LIN {X 0,Y 466.236,Z 937.259,A -85,B 0,C 180,E1 20114.358,E2 20114.358} C_VEL
LIN {X 0,Y 461.421,Z 960.105,A -85,B 0,C 180,E1 20112.986,E2 20112.986} C_VEL
LIN {X 0,Y 456.989,Z 979.325,A -85,B 0,C 180,E1 20111.61,E2 20111.61} C_VEL
LIN {X 0,Y 451.374,Z 1001.605,A -85,B 0,C 180,E1 20109.724,E2 20109.724} C_VEL
LIN {X 0,Y 446.55,Z 1019.671,A -85,B 0,C 180,E1 20107.926,E2 20107.926} C_VEL
LIN {X 0,Y 441.064,Z 1039.324,A -85,B 0,C 180,E1 20105.635,E2 20105.635} C_VEL
LIN {X 0,Y 436.572,Z 1055.083,A -85,B 0,C 180,E1 20103.502,E2 20103.502} C_VEL
LIN {X 0,Y 431.661,Z 1072.275,A -85,B 0,C 180,E1 20100.792,E2 20100.792} C_VEL
LIN {X 0,Y 427.908,Z 1085.783,A -85,B 0,C 180,E1 20098.317,E2 20098.317} C_VEL
LIN {X 0,Y 424.121,Z 1100.061,A -85,B 0,C 180,E1 20095.26,E2 20095.26} C_VEL
LIN {X 0,Y 421.416,Z 1111.21,A -85,B 0,C 180,E1 20092.458,E2 20092.458} C_VEL
LIN {X 0,Y 419.039,Z 1122.409,A -85,B 0,C 180,E1 20089.105,E2 20089.105} C_VEL
LIN {X 0,Y 417.651,Z 1130.324,A -85,B 0,C 180,E1 20086.254,E2 20086.254} C_VEL
LIN {X 0,Y 416.596,Z 1138.166,A -85,B 0,C 180,E1 20082.757,E2 20082.757} C_VEL
LIN {X 0,Y 416.157,Z 1143.104,A -85,B 0,C 180,E1 20079.902,E2 20079.902} C_VEL
LIN {X 0,Y 415.971,Z 1147.181,A -85,B 0,C 180,E1 20076.764,E2 20076.764} C_VEL
LIN {X 0,Y 415.942,Z 1149.613,A -85,B 0,C 180,E1 20073.583,E2 20073.583} C_VEL
LIN {X 0,Y 415.943,Z 1150.522,A -85,B 0,C 180,E1 20070.964,E2 20070.964} C_VEL
LIN {X 0,Y 415.947,Z 1150.354,A -85,B 0,C 180,E1 20068.071,E2 20068.071} C_VEL
LIN {X 0,Y 415.927,Z 1148.612,A -85,B 0,C 180,E1 20064.897,E2 20064.897} C_VEL
LIN {X 0,Y 415.991,Z 1145.845,A -85,B 0,C 180,E1 20062.125,E2 20062.125} C_VEL
LIN {X 0,Y 416.258,Z 1141.713,A -85,B 0,C 180,E1 20059.201,E2 20059.201} C_VEL
LIN {X 0,Y 416.938,Z 1135.233,A -85,B 0,C 180,E1 20055.841,E2 20055.841} C_VEL
LIN {X 0,Y 417.947,Z 1128.442,A -85,B 0,C 180,E1 20053.03,E2 20053.03} C_VEL
LIN {X 0,Y 419.816,Z 1118.491,A -85,B 0,C 180,E1 20049.651,E2 20049.651} C_VEL
LIN {X 0,Y 422.069,Z 1108.405,A -85,B 0,C 180,E1 20046.807,E2 20046.807} C_VEL
LIN {X 0,Y 425.401,Z 1095.098,A -85,B 0,C 180,E1 20043.625,E2 20043.625} C_VEL
LIN {X 0,Y 428.676,Z 1082.856,A -85,B 0,C 180,E1 20041.129,E2 20041.129} C_VEL
LIN {X 0,Y 433.056,Z 1067.359,A -85,B 0,C 180,E1 20038.39,E2 20038.39} C_VEL
LIN {X 0,Y 437.389,Z 1052.082,A -85,B 0,C 180,E1 20036.082,E2 20036.082} C_VEL
LIN {X 0,Y 442.334,Z 1034.815,A -85,B 0,C 180,E1 20033.804,E2 20033.804} C_VEL
LIN {X 0,Y 447.361,Z 1016.456,A -85,B 0,C 180,E1 20031.748,E2 20031.748} C_VEL
LIN {X 0,Y 452.648,Z 996.689,A -85,B 0,C 180,E1 20029.832,E2 20029.832} C_VEL
LIN {X 0,Y 457.714,Z 976.039,A -85,B 0,C 180,E1 20028.153,E2 20028.153} C_VEL
LIN {X 0,Y 462.616,Z 954.653,A -85,B 0,C 180,E1 20026.667,E2 20026.667} C_VEL
LIN {X 0,Y 466.859,Z 933.595,A -85,B 0,C 180,E1 20025.459,E2 20025.459} C_VEL
LIN {X 0,Y 470.626,Z 912.697,A -85,B 0,C 180,E1 20024.449,E2 20024.449} C_VEL
LIN {X 0,Y 474.229,Z 888.902,A -85,B 0,C 180,E1 20023.533,E2 20023.533} C_VEL
LIN {X 0,Y 476.825,Z 868.071,A -85,B 0,C 180,E1 20022.903,E2 20022.903} C_VEL
LIN {X 0,Y 479.197,Z 841.622,A -85,B 0,C 180,E1 20022.311,E2 20022.311} C_VEL
LIN {X 0,Y 490.289,Z 617.268,A -85,B 0,C 180,E1 20018.698,E2 20018.698} C_VEL
LIN {X 0,Y 493.313,Z 555.727,A -85,B 0,C 180,E1 20017.706,E2 20017.706} C_VEL
LIN {X 0,Y 483.018,Z 538.654,A -85,B 0,C 180,E1 20015.789,E2 20015.789} C_VEL
LIN {X 0,Y 473.224,Z 523.488,A -85,B 0,C 180,E1 20013.832,E2 20013.832} C_VEL
LIN {X 0,Y 462.632,Z 508.305,A -85,B 0,C 180,E1 20011.536,E2 20011.536} C_VEL
LIN {X 0,Y 453.738,Z 496.412,A -85,B 0,C 180,E1 20009.434,E2 20009.434} C_VEL
LIN {X 0,Y 446.328,Z 486.795,A -85,B 0,C 180,E1 20007.52,E2 20007.52} C_VEL
LIN {X 0,Y 441.143,Z 480.531,A -85,B 0,C 180,E1 20006.086,E2 20006.086} C_VEL
LIN {X 0,Y 436.301,Z 474.731,A -85,B 0,C 180,E1 20004.652,E2 20004.652} C_VEL
LIN {X 0,Y 431.339,Z 468.954,A -85,B 0,C 180,E1 20003.064,E2 20003.064} C_VEL
LIN {X 0,Y 429.525,Z 465.262,A -85,B 0,C 180,E1 20001.724,E2 20001.724} C_VEL
LIN {X 0,Y 427.505,Z 461.609,A -85,B 0,C 180,E1 20000.11,E2 20000.11} C_VEL
LIN {X 0,Y 426.506,Z 459.96,A -85,B 0,C 180,E1 19999.303,E2 19999.303} C_VEL
LIN {X 0,Y 424.096,Z 455.355,A -85,B 0,C 180,E1 19996.999,E2 19996.999} C_VEL
LIN {X 0,Y 421.764,Z 451.295,A -85,B 0,C 180,E1 19994.554,E2 19994.554} C_VEL
LIN {X 0,Y 421.091,Z 450.043,A -85,B 0,C 180,E1 19993.736,E2 19993.736} C_VEL
LIN {X 0,Y 418.609,Z 445.587,A -85,B 0,C 180,E1 19990.181,E2 19990.181} C_VEL
LIN {X 0,Y 418.499,Z 445.082,A -85,B 0,C 180,E1 19988.657,E2 19988.657} C_VEL
LIN {X 0,Y 418.484,Z 445.068,A -85,B 0,C 180,E1 19984.897,E2 19984.897} C_VEL
LIN {X 0,Y 418.484,Z 445.066,A -85,B 0,C 180,E1 19981.095,E2 19981.095} C_VEL
LIN {X 0,Y 418.501,Z 445.072,A -85,B 0,C 180,E1 19977.398,E2 19977.398} C_VEL
LIN {X 0,Y 418.519,Z 445.085,A -85,B 0,C 180,E1 19973.553,E2 19973.553} C_VEL
LIN {X 0,Y 418.524,Z 445.143,A -85,B 0,C 180,E1 19969.678,E2 19969.678} C_VEL
LIN {X 0,Y 418.601,Z 445.836,A -85,B 0,C 180,E1 19968.704,E2 19968.704} C_VEL
LIN {X 0,Y 421.63,Z 451.075,A -85,B 0,C 180,E1 19964.597,E2 19964.597} C_VEL
LIN {X 0,Y 423.884,Z 455.148,A -85,B 0,C 180,E1 19962.142,E2 19962.142} C_VEL
LIN {X 0,Y 424.578,Z 456.381,A -85,B 0,C 180,E1 19961.462,E2 19961.462} C_VEL
LIN {X 0,Y 426.442,Z 459.915,A -85,B 0,C 180,E1 19959.695,E2 19959.695} C_VEL
LIN {X 0,Y 427.478,Z 462.022,A -85,B 0,C 180,E1 19958.743,E2 19958.743} C_VEL
LIN {X 0,Y 429.853,Z 466.303,A -85,B 0,C 180,E1 19956.851,E2 19956.851} C_VEL
LIN {X 0,Y 432.472,Z 471.575,A -85,B 0,C 180,E1 19954.823,E2 19954.823} C_VEL
LIN {X 0,Y 434.744,Z 476.119,A -85,B 0,C 180,E1 19953.205,E2 19953.205} C_VEL
LIN {X 0,Y 437.115,Z 481.055,A -85,B 0,C 180,E1 19951.589,E2 19951.589} C_VEL
LIN {X 0,Y 439.13,Z 484.762,A -85,B 0,C 180,E1 19950.502,E2 19950.502} C_VEL
LIN {X 0,Y 446.478,Z 494.703,A -85,B 0,C 180,E1 19948.434,E2 19948.434} C_VEL
LIN {X 0,Y 452.479,Z 502.886,A -85,B 0,C 180,E1 19946.885,E2 19946.885} C_VEL
LIN {X 0,Y 461.013,Z 515.147,A -85,B 0,C 180,E1 19944.841,E2 19944.841} C_VEL
LIN {X 0,Y 469.958,Z 528.922,A -85,B 0,C 180,E1 19942.864,E2 19942.864} C_VEL
LIN {X 0,Y 479.843,Z 544.931,A -85,B 0,C 180,E1 19940.847,E2 19940.847} C_VEL
LIN {X 0,Y 489.836,Z 562.594,A -85,B 0,C 180,E1 19938.945,E2 19938.945} C_VEL
LIN {X 0,Y 490.651,Z 564.525,A -85,B 0,C 180,E1 19938.786,E2 19938.786} C_VEL
LIN {X 0,Y 491.161,Z 569.373,A -85,B 0,C 180,E1 19938.607,E2 19938.607} C_VEL
LIN {X 0,Y 479.889,Z 824.745,A -85,B 0,C 180,E1 19934.734,E2 19934.734} C_VEL
LIN {X 0,Y 478.092,Z 855.335,A -85,B 0,C 180,E1 19934.21,E2 19934.21} C_VEL
LIN {X 0,Y 475.844,Z 877.482,A -85,B 0,C 180,E1 19933.668,E2 19933.668} C_VEL
LIN {X 0,Y 472.694,Z 900.618,A -85,B 0,C 180,E1 19932.891,E2 19932.891} C_VEL
LIN {X 0,Y 469.116,Z 922.276,A -85,B 0,C 180,E1 19931.966,E2 19931.966} C_VEL
LIN {X 0,Y 464.908,Z 943.457,A -85,B 0,C 180,E1 19930.831,E2 19930.831} C_VEL
LIN {X 0,Y 460.365,Z 963.847,A -85,B 0,C 180,E1 19929.523,E2 19929.523} C_VEL
LIN {X 0,Y 455.443,Z 983.36,A -85,B 0,C 180,E1 19928.003,E2 19928.003} C_VEL
LIN {X 0,Y 450.456,Z 1001.908,A -85,B 0,C 180,E1 19926.316,E2 19926.316} C_VEL
LIN {X 0,Y 445.221,Z 1019.736,A -85,B 0,C 180,E1 19924.38,E2 19924.38} C_VEL
LIN {X 0,Y 440.166,Z 1036.473,A -85,B 0,C 180,E1 19922.265,E2 19922.265} C_VEL
LIN {X 0,Y 435.489,Z 1051.384,A -85,B 0,C 180,E1 19920.035,E2 19920.035} C_VEL
LIN {X 0,Y 430.926,Z 1065.976,A -85,B 0,C 180,E1 19917.5,E2 19917.5} C_VEL
LIN {X 0,Y 427.066,Z 1078.461,A -85,B 0,C 180,E1 19914.925,E2 19914.925} C_VEL
LIN {X 0,Y 423.388,Z 1091.027,A -85,B 0,C 180,E1 19911.855,E2 19911.855} C_VEL
LIN {X 0,Y 420.871,Z 1100.299,A -85,B 0,C 180,E1 19909.139,E2 19909.139} C_VEL
LIN {X 0,Y 418.723,Z 1109.293,A -85,B 0,C 180,E1 19905.939,E2 19905.939} C_VEL
LIN {X 0,Y 417.417,Z 1115.919,A -85,B 0,C 180,E1 19903.013,E2 19903.013} C_VEL
LIN {X 0,Y 416.528,Z 1121.699,A -85,B 0,C 180,E1 19899.674,E2 19899.674} C_VEL
LIN {X 0,Y 416.151,Z 1125.344,A -85,B 0,C 180,E1 19896.761,E2 19896.761} C_VEL
LIN {X 0,Y 415.984,Z 1127.881,A -85,B 0,C 180,E1 19893.445,E2 19893.445} C_VEL
LIN {X 0,Y 415.96,Z 1128.751,A -85,B 0,C 180,E1 19890.689,E2 19890.689} C_VEL
LIN {X 0,Y 415.97,Z 1128.859,A -85,B 0,C 180,E1 19889.97,E2 19889.97} C_VEL
LIN {X 0,Y 414.938,Z 1128.793,A -85,B 0,C 180,E1 19888.908,E2 19888.908} C_VEL
LIN {X 0,Y 408.532,Z 1127.889,A -85,B 0,C 180,E1 19885.92,E2 19885.92} C_VEL
LIN {X 0,Y 408.028,Z 1127.363,A -85,B 0,C 180,E1 19885.143,E2 19885.143} C_VEL
LIN {X 0,Y 408.249,Z 1124.747,A -85,B 0,C 180,E1 19882.258,E2 19882.258} C_VEL
LIN {X 0,Y 408.8,Z 1120.397,A -85,B 0,C 180,E1 19879.002,E2 19879.002} C_VEL
LIN {X 0,Y 409.823,Z 1114.59,A -85,B 0,C 180,E1 19875.878,E2 19875.878} C_VEL
LIN {X 0,Y 411.56,Z 1106.902,A -85,B 0,C 180,E1 19872.613,E2 19872.613} C_VEL
LIN {X 0,Y 413.856,Z 1098.115,A -85,B 0,C 180,E1 19869.624,E2 19869.624} C_VEL
LIN {X 0,Y 417.224,Z 1086.65,A -85,B 0,C 180,E1 19866.408,E2 19866.408} C_VEL
LIN {X 0,Y 420.762,Z 1075.415,A -85,B 0,C 180,E1 19863.768,E2 19863.768} C_VEL
LIN {X 0,Y 425.294,Z 1061.422,A -85,B 0,C 180,E1 19860.997,E2 19860.997} C_VEL
LIN {X 0,Y 430.002,Z 1047.109,A -85,B 0,C 180,E1 19858.583,E2 19858.583} C_VEL
LIN {X 0,Y 435.22,Z 1030.861,A -85,B 0,C 180,E1 19856.271,E2 19856.271} C_VEL
LIN {X 0,Y 440.64,Z 1013.592,A -85,B 0,C 180,E1 19854.165,E2 19854.165} C_VEL
LIN {X 0,Y 446.057,Z 994.989,A -85,B 0,C 180,E1 19852.268,E2 19852.268} C_VEL
LIN {X 0,Y 451.521,Z 974.977,A -85,B 0,C 180,E1 19850.538,E2 19850.538} C_VEL
LIN {X 0,Y 456.076,Z 956.544,A -85,B 0,C 180,E1 19849.207,E2 19849.207} C_VEL
LIN {X 0,Y 460.892,Z 934.937,A -85,B 0,C 180,E1 19847.899,E2 19847.899} C_VEL
LIN {X 0,Y 464.708,Z 914.889,A -85,B 0,C 180,E1 19846.909,E2 19846.909} C_VEL
LIN {X 0,Y 468.44,Z 891.824,A -85,B 0,C 180,E1 19845.995,E2 19845.995} C_VEL
LIN {X 0,Y 471.082,Z 870.943,A -85,B 0,C 180,E1 19845.361,E2 19845.361} C_VEL
LIN {X 0,Y 473.346,Z 846.549,A -85,B 0,C 180,E1 19844.819,E2 19844.819} C_VEL
LIN {X 0,Y 481.939,Z 658.642,A -85,B 0,C 180,E1 19841.926,E2 19841.926} C_VEL
LIN {X 0,Y 486.071,Z 569.379,A -85,B 0,C 180,E1 19840.545,E2 19840.545} C_VEL
LIN {X 0,Y 485.457,Z 567.538,A -85,B 0,C 180,E1 19840.413,E2 19840.413} C_VEL
LIN {X 0,Y 475.186,Z 549.156,A -85,B 0,C 180,E1 19838.39,E2 19838.39} C_VEL
LIN {X 0,Y 463.604,Z 530.342,A -85,B 0,C 180,E1 19835.919,E2 19835.919} C_VEL
LIN {X 0,Y 451.846,Z 512.633,A -85,B 0,C 180,E1 19833.133,E2 19833.133} C_VEL
LIN {X 0,Y 445.276,Z 503.579,A -85,B 0,C 180,E1 19831.431,E2 19831.431} C_VEL
LIN {X 0,Y 438.875,Z 494.83,A -85,B 0,C 180,E1 19829.63,E2 19829.63} C_VEL
LIN {X 0,Y 434.964,Z 489.644,A -85,B 0,C 180,E1 19828.452,E2 19828.452} C_VEL
LIN {X 0,Y 429.781,Z 482.666,A -85,B 0,C 180,E1 19826.681,E2 19826.681} C_VEL
LIN {X 0,Y 428.07,Z 479.202,A -85,B 0,C 180,E1 19825.454,E2 19825.454} C_VEL
LIN {X 0,Y 426.124,Z 475.201,A -85,B 0,C 180,E1 19823.95,E2 19823.95} C_VEL
LIN {X 0,Y 423.943,Z 470.874,A -85,B 0,C 180,E1 19822.171,E2 19822.171} C_VEL
LIN {X 0,Y 421.585,Z 466.288,A -85,B 0,C 180,E1 19820.08,E2 19820.08} C_VEL
LIN {X 0,Y 419.645,Z 462.586,A -85,B 0,C 180,E1 19818.188,E2 19818.188} C_VEL
LIN {X 0,Y 416.217,Z 456.382,A -85,B 0,C 180,E1 19814.326,E2 19814.326} C_VEL
LIN {X 0,Y 413.397,Z 451.317,A -85,B 0,C 180,E1 19810.029,E2 19810.029} C_VEL
LIN {X 0,Y 410.952,Z 447.698,A -85,B 0,C 180,E1 19803.987,E2 19803.987} C_VEL
LIN {X 0,Y 410.734,Z 446.955,A -85,B 0,C 180,E1 19800.418,E2 19800.418} C_VEL
LIN {X 0,Y 410.903,Z 447.66,A -85,B 0,C 180,E1 19797.071,E2 19797.071} C_VEL
LIN {X 0,Y 412.969,Z 450.874,A -85,B 0,C 180,E1 19791.507,E2 19791.507} C_VEL
LIN {X 0,Y 413.909,Z 452.207,A -85,B 0,C 180,E1 19789.983,E2 19789.983} C_VEL
LIN {X 0,Y 416.606,Z 456.731,A -85,B 0,C 180,E1 19786.254,E2 19786.254} C_VEL
LIN {X 0,Y 419.083,Z 461.489,A -85,B 0,C 180,E1 19783.363,E2 19783.363} C_VEL
LIN {X 0,Y 420.011,Z 463.276,A -85,B 0,C 180,E1 19782.402,E2 19782.402} C_VEL
LIN {X 0,Y 422.459,Z 467.556,A -85,B 0,C 180,E1 19780.217,E2 19780.217} C_VEL
LIN {X 0,Y 423.625,Z 469.957,A -85,B 0,C 180,E1 19779.337,E2 19779.337} C_VEL
LIN {X 0,Y 427.225,Z 474.003,A -85,B 0,C 180,E1 19778.008,E2 19778.008} C_VEL
LIN {X 0,Y 432.384,Z 480.06,A -85,B 0,C 180,E1 19776.273,E2 19776.273} C_VEL
LIN {X 0,Y 436.767,Z 485.289,A -85,B 0,C 180,E1 19774.907,E2 19774.907} C_VEL
LIN {X 0,Y 441.245,Z 490.776,A -85,B 0,C 180,E1 19773.595,E2 19773.595} C_VEL
LIN {X 0,Y 446.228,Z 497.114,A -85,B 0,C 180,E1 19772.22,E2 19772.22} C_VEL
LIN {X 0,Y 454.022,Z 507.317,A -85,B 0,C 180,E1 19770.223,E2 19770.223} C_VEL
LIN {X 0,Y 463.425,Z 520.432,A -85,B 0,C 180,E1 19768.015,E2 19768.015} C_VEL
LIN {X 0,Y 474.721,Z 537.249,A -85,B 0,C 180,E1 19765.597,E2 19765.597} C_VEL
LIN {X 0,Y 487.154,Z 557.652,A -85,B 0,C 180,E1 19763.159,E2 19763.159} C_VEL
LIN {X 0,Y 488.226,Z 559.815,A -85,B 0,C 180,E1 19762.951,E2 19762.951} C_VEL
LIN {X 0,Y 476.442,Z 790.275,A -85,B 0,C 180,E1 19759.246,E2 19759.246} C_VEL
LIN {X 0,Y 473.431,Z 846.64,A -85,B 0,C 180,E1 19758.306,E2 19758.306} C_VEL
LIN {X 0,Y 470.957,Z 870.988,A -85,B 0,C 180,E1 19757.723,E2 19757.723} C_VEL
LIN {X 0,Y 467.992,Z 893.628,A -85,B 0,C 180,E1 19757.011,E2 19757.011} C_VEL
LIN {X 0,Y 464.181,Z 916.79,A -85,B 0,C 180,E1 19756.064,E2 19756.064} C_VEL
LIN {X 0,Y 460.216,Z 937.876,A -85,B 0,C 180,E1 19755.008,E2 19755.008} C_VEL
LIN {X 0,Y 455.197,Z 960.834,A -85,B 0,C 180,E1 19753.61,E2 19753.61} C_VEL
LIN {X 0,Y 450.466,Z 980.654,A -85,B 0,C 180,E1 19752.171,E2 19752.171} C_VEL
LIN {X 0,Y 444.882,Z 1001.936,A -85,B 0,C 180,E1 19750.338,E2 19750.338} C_VEL
LIN {X 0,Y 439.892,Z 1019.961,A -85,B 0,C 180,E1 19748.522,E2 19748.522} C_VEL
LIN {X 0,Y 434.358,Z 1039.027,A -85,B 0,C 180,E1 19746.272,E2 19746.272} C_VEL
LIN {X 0,Y 429.514,Z 1055.379,A -85,B 0,C 180,E1 19744.029,E2 19744.029} C_VEL
LIN {X 0,Y 424.544,Z 1072.008,A -85,B 0,C 180,E1 19741.366,E2 19741.366} C_VEL
LIN {X 0,Y 420.613,Z 1085.524,A -85,B 0,C 180,E1 19738.854,E2 19738.854} C_VEL
LIN {X 0,Y 416.631,Z 1099.816,A -85,B 0,C 180,E1 19735.747,E2 19735.747} C_VEL
LIN {X 0,Y 413.783,Z 1110.97,A -85,B 0,C 180,E1 19732.896,E2 19732.896} C_VEL
LIN {X 0,Y 411.246,Z 1122.249,A -85,B 0,C 180,E1 19729.457,E2 19729.457} C_VEL
LIN {X 0,Y 409.785,Z 1130.065,A -85,B 0,C 180,E1 19726.588,E2 19726.588} C_VEL
LIN {X 0,Y 408.651,Z 1137.946,A -85,B 0,C 180,E1 19723.009,E2 19723.009} C_VEL
LIN {X 0,Y 408.18,Z 1142.796,A -85,B 0,C 180,E1 19720.159,E2 19720.159} C_VEL
LIN {X 0,Y 407.982,Z 1146.872,A -85,B 0,C 180,E1 19716.98,E2 19716.98} C_VEL
LIN {X 0,Y 407.946,Z 1149.331,A -85,B 0,C 180,E1 19713.795,E2 19713.795} C_VEL
LIN {X 0,Y 407.95,Z 1150.289,A -85,B 0,C 180,E1 19711.124,E2 19711.124} C_VEL
LIN {X 0,Y 407.95,Z 1150.216,A -85,B 0,C 180,E1 19708.455,E2 19708.455} C_VEL
LIN {X 0,Y 407.934,Z 1148.754,A -85,B 0,C 180,E1 19705.22,E2 19705.22} C_VEL
LIN {X 0,Y 407.982,Z 1145.962,A -85,B 0,C 180,E1 19702.253,E2 19702.253} C_VEL
LIN {X 0,Y 408.228,Z 1142.139,A -85,B 0,C 180,E1 19699.415,E2 19699.415} C_VEL
LIN {X 0,Y 408.9,Z 1135.95,A -85,B 0,C 180,E1 19695.99,E2 19695.99} C_VEL
LIN {X 0,Y 409.979,Z 1128.861,A -85,B 0,C 180,E1 19692.949,E2 19692.949} C_VEL
LIN {X 0,Y 411.794,Z 1119.671,A -85,B 0,C 180,E1 19689.682,E2 19689.682} C_VEL
LIN {X 0,Y 414.17,Z 1109.348,A -85,B 0,C 180,E1 19686.676,E2 19686.676} C_VEL
LIN {X 0,Y 417.349,Z 1097.231,A -85,B 0,C 180,E1 19683.642,E2 19683.642} C_VEL
LIN {X 0,Y 421.006,Z 1084.029,A -85,B 0,C 180,E1 19680.864,E2 19680.864} C_VEL
LIN {X 0,Y 425.266,Z 1069.575,A -85,B 0,C 180,E1 19678.219,E2 19678.219} C_VEL
LIN {X 0,Y 430.084,Z 1053.293,A -85,B 0,C 180,E1 19675.682,E2 19675.682} C_VEL
LIN {X 0,Y 434.968,Z 1036.862,A -85,B 0,C 180,E1 19673.46,E2 19673.46} C_VEL
LIN {X 0,Y 440.387,Z 1017.978,A -85,B 0,C 180,E1 19671.28,E2 19671.28} C_VEL
LIN {X 0,Y 445.24,Z 1000.431,A -85,B 0,C 180,E1 19669.532,E2 19669.532} C_VEL
LIN {X 0,Y 450.867,Z 978.743,A -85,B 0,C 180,E1 19667.695,E2 19667.695} C_VEL
LIN {X 0,Y 455.394,Z 959.724,A -85,B 0,C 180,E1 19666.327,E2 19666.327} C_VEL
LIN {X 0,Y 460.414,Z 936.48,A -85,B 0,C 180,E1 19664.929,E2 19664.929} C_VEL
LIN {X 0,Y 464.258,Z 915.95,A -85,B 0,C 180,E1 19663.908,E2 19663.908} C_VEL
LIN {X 0,Y 468.237,Z 891.258,A -85,B 0,C 180,E1 19662.919,E2 19662.919} C_VEL
LIN {X 0,Y 470.981,Z 870.101,A -85,B 0,C 180,E1 19662.263,E2 19662.263} C_VEL
LIN {X 0,Y 473.431,Z 845.26,A -85,B 0,C 180,E1 19661.679,E2 19661.679} C_VEL
LIN {X 0,Y 477.17,Z 773.846,A -85,B 0,C 180,E1 19660.498,E2 19660.498} C_VEL
LIN {X 0,Y 488.114,Z 559.467,A -85,B 0,C 180,E1 19657.05,E2 19657.05} C_VEL
LIN {X 0,Y 476.77,Z 540.614,A -85,B 0,C 180,E1 19654.855,E2 19654.855} C_VEL
LIN {X 0,Y 466.825,Z 525.484,A -85,B 0,C 180,E1 19652.777,E2 19652.777} C_VEL
LIN {X 0,Y 456.774,Z 511.022,A -85,B 0,C 180,E1 19650.485,E2 19650.485} C_VEL
LIN {X 0,Y 447.495,Z 498.7,A -85,B 0,C 180,E1 19648.166,E2 19648.166} C_VEL
LIN {X 0,Y 439.334,Z 488.324,A -85,B 0,C 180,E1 19645.911,E2 19645.911} C_VEL
LIN {X 0,Y 433.643,Z 481.552,A -85,B 0,C 180,E1 19644.196,E2 19644.196} C_VEL
LIN {X 0,Y 428.84,Z 475.886,A -85,B 0,C 180,E1 19642.626,E2 19642.626} C_VEL
LIN {X 0,Y 425.089,Z 471.586,A -85,B 0,C 180,E1 19641.31,E2 19641.31} C_VEL
LIN {X 0,Y 422.894,Z 468.789,A -85,B 0,C 180,E1 19640.339,E2 19640.339} C_VEL
LIN {X 0,Y 421.848,Z 466.525,A -85,B 0,C 180,E1 19639.375,E2 19639.375} C_VEL
LIN {X 0,Y 419.726,Z 462.397,A -85,B 0,C 180,E1 19637.324,E2 19637.324} C_VEL
LIN {X 0,Y 416.96,Z 457.656,A -85,B 0,C 180,E1 19634.442,E2 19634.442} C_VEL
LIN {X 0,Y 416.288,Z 456.416,A -85,B 0,C 180,E1 19633.615,E2 19633.615} C_VEL
LIN {X 0,Y 413.474,Z 451.36,A -85,B 0,C 180,E1 19629.465,E2 19629.465} C_VEL
LIN {X 0,Y 410.866,Z 447.487,A -85,B 0,C 180,E1 19623.348,E2 19623.348} C_VEL
LIN {X 0,Y 410.683,Z 446.579,A -85,B 0,C 180,E1 19619.86,E2 19619.86} C_VEL
LIN {X 0,Y 410.796,Z 447.248,A -85,B 0,C 180,E1 19616.232,E2 19616.232} C_VEL
LIN {X 0,Y 412.43,Z 450.304,A -85,B 0,C 180,E1 19611.074,E2 19611.074} C_VEL
LIN {X 0,Y 413.759,Z 451.952,A -85,B 0,C 180,E1 19608.994,E2 19608.994} C_VEL
LIN {X 0,Y 416.829,Z 457.521,A -85,B 0,C 180,E1 19604.649,E2 19604.649} C_VEL
LIN {X 0,Y 419.209,Z 461.669,A -85,B 0,C 180,E1 19602.08,E2 19602.08} C_VEL
LIN {X 0,Y 421.569,Z 466.252,A -85,B 0,C 180,E1 19599.739,E2 19599.739} C_VEL
LIN {X 0,Y 424.757,Z 472.41,A -85,B 0,C 180,E1 19596.989,E2 19596.989} C_VEL
LIN {X 0,Y 427.331,Z 477.665,A -85,B 0,C 180,E1 19594.943,E2 19594.943} C_VEL
LIN {X 0,Y 429.595,Z 482.246,A -85,B 0,C 180,E1 19593.307,E2 19593.307} C_VEL
LIN {X 0,Y 431.567,Z 485.164,A -85,B 0,C 180,E1 19592.469,E2 19592.469} C_VEL
LIN {X 0,Y 437.443,Z 493.007,A -85,B 0,C 180,E1 19590.64,E2 19590.64} C_VEL
LIN {X 0,Y 443.691,Z 501.448,A -85,B 0,C 180,E1 19588.856,E2 19588.856} C_VEL
LIN {X 0,Y 449.505,Z 509.486,A -85,B 0,C 180,E1 19587.318,E2 19587.318} C_VEL
LIN {X 0,Y 458.139,Z 522.121,A -85,B 0,C 180,E1 19585.199,E2 19585.199} C_VEL
LIN {X 0,Y 466.687,Z 535.452,A -85,B 0,C 180,E1 19583.267,E2 19583.267} C_VEL
LIN {X 0,Y 476.309,Z 551.29,A -85,B 0,C 180,E1 19581.256,E2 19581.256} C_VEL
LIN {X 0,Y 485.816,Z 568.322,A -85,B 0,C 180,E1 19579.4,E2 19579.4} C_VEL
LIN {X 0,Y 485.988,Z 571.508,A -85,B 0,C 180,E1 19579.303,E2 19579.303} C_VEL
LIN {X 0,Y 474.351,Z 825.865,A -85,B 0,C 180,E1 19575.418,E2 19575.418} C_VEL
LIN {X 0,Y 472.525,Z 855.575,A -85,B 0,C 180,E1 19574.903,E2 19574.903} C_VEL
LIN {X 0,Y 470.2,Z 877.799,A -85,B 0,C 180,E1 19574.355,E2 19574.355} C_VEL
LIN {X 0,Y 467.002,Z 900.564,A -85,B 0,C 180,E1 19573.585,E2 19573.585} C_VEL
LIN {X 0,Y 463.329,Z 922.167,A -85,B 0,C 180,E1 19572.659,E2 19572.659} C_VEL
LIN {X 0,Y 459.017,Z 943.271,A -85,B 0,C 180,E1 19571.524,E2 19571.524} C_VEL
LIN {X 0,Y 454.345,Z 963.629,A -85,B 0,C 180,E1 19570.212,E2 19570.212} C_VEL
LIN {X 0,Y 449.331,Z 982.931,A -85,B 0,C 180,E1 19568.705,E2 19568.705} C_VEL
LIN {X 0,Y 444.041,Z 1001.994,A -85,B 0,C 180,E1 19566.958,E2 19566.958} C_VEL
LIN {X 0,Y 438.58,Z 1019.974,A -85,B 0,C 180,E1 19564.986,E2 19564.986} C_VEL
LIN {X 0,Y 433.312,Z 1036.753,A -85,B 0,C 180,E1 19562.839,E2 19562.839} C_VEL
LIN {X 0,Y 428.366,Z 1051.938,A -85,B 0,C 180,E1 19560.535,E2 19560.535} C_VEL
LIN {X 0,Y 423.475,Z 1066.914,A -85,B 0,C 180,E1 19557.873,E2 19557.873} C_VEL
LIN {X 0,Y 419.677,Z 1078.709,A -85,B 0,C 180,E1 19555.395,E2 19555.395} C_VEL
LIN {X 0,Y 415.878,Z 1091.075,A -85,B 0,C 180,E1 19552.326,E2 19552.326} C_VEL
LIN {X 0,Y 413.18,Z 1100.531,A -85,B 0,C 180,E1 19549.509,E2 19549.509} C_VEL
LIN {X 0,Y 410.909,Z 1109.518,A -85,B 0,C 180,E1 19546.251,E2 19546.251} C_VEL
LIN {X 0,Y 409.521,Z 1116.14,A -85,B 0,C 180,E1 19543.268,E2 19543.268} C_VEL
LIN {X 0,Y 408.575,Z 1121.915,A -85,B 0,C 180,E1 19539.864,E2 19539.864} C_VEL
LIN {X 0,Y 408.167,Z 1125.558,A -85,B 0,C 180,E1 19536.894,E2 19536.894} C_VEL
LIN {X 0,Y 407.988,Z 1128.092,A -85,B 0,C 180,E1 19533.513,E2 19533.513} C_VEL
LIN {X 0,Y 407.963,Z 1128.961,A -85,B 0,C 180,E1 19530.702,E2 19530.702} C_VEL
LIN {X 0,Y 407.972,Z 1128.596,A -85,B 0,C 180,E1 19527.472,E2 19527.472} C_VEL
LIN {X 0,Y 408.028,Z 1127.363,A -85,B 0,C 180,E1 19525.143,E2 19525.143} C_VEL
LIN {X 0,Y 407.087,Z 1126.577,A -85,B 0,C 180,E1 19524.066,E2 19524.066} C_VEL
LIN {X 0,Y 400.941,Z 1123.752,A -85,B 0,C 180,E1 19521.035,E2 19521.035} C_VEL
LIN {X 0,Y 400.541,Z 1122.704,A -85,B 0,C 180,E1 19520.252,E2 19520.252} C_VEL
LIN {X 0,Y 401.391,Z 1117.669,A -85,B 0,C 180,E1 19517.044,E2 19517.044} C_VEL
LIN {X 0,Y 402.89,Z 1110.666,A -85,B 0,C 180,E1 19513.713,E2 19513.713} C_VEL
LIN {X 0,Y 405.078,Z 1102.402,A -85,B 0,C 180,E1 19510.535,E2 19510.535} C_VEL
LIN {X 0,Y 407.934,Z 1092.652,A -85,B 0,C 180,E1 19507.519,E2 19507.519} C_VEL
LIN {X 0,Y 411.619,Z 1081.236,A -85,B 0,C 180,E1 19504.535,E2 19504.535} C_VEL
LIN {X 0,Y 415.681,Z 1069.001,A -85,B 0,C 180,E1 19501.87,E2 19501.87} C_VEL
LIN {X 0,Y 420.508,Z 1054.969,A -85,B 0,C 180,E1 19499.254,E2 19499.254} C_VEL
LIN {X 0,Y 425.415,Z 1040.367,A -85,B 0,C 180,E1 19496.955,E2 19496.955} C_VEL
LIN {X 0,Y 430.931,Z 1023.738,A -85,B 0,C 180,E1 19494.707,E2 19494.707} C_VEL
LIN {X 0,Y 436.28,Z 1006.72,A -85,B 0,C 180,E1 19492.767,E2 19492.767} C_VEL
LIN {X 0,Y 442.081,Z 987.161,A -85,B 0,C 180,E1 19490.873,E2 19490.873} C_VEL
LIN {X 0,Y 447.016,Z 968.938,A -85,B 0,C 180,E1 19489.389,E2 19489.389} C_VEL
LIN {X 0,Y 452.393,Z 947.06,A -85,B 0,C 180,E1 19487.902,E2 19487.902} C_VEL
LIN {X 0,Y 456.631,Z 927.356,A -85,B 0,C 180,E1 19486.797,E2 19486.797} C_VEL
LIN {X 0,Y 460.923,Z 903.891,A -85,B 0,C 180,E1 19485.735,E2 19485.735} C_VEL
LIN {X 0,Y 464.19,Z 882.173,A -85,B 0,C 180,E1 19484.965,E2 19484.965} C_VEL
LIN {X 0,Y 466.866,Z 858.532,A -85,B 0,C 180,E1 19484.346,E2 19484.346} C_VEL
LIN {X 0,Y 468.623,Z 834.837,A -85,B 0,C 180,E1 19483.901,E2 19483.901} C_VEL
LIN {X 0,Y 480.564,Z 582.416,A -85,B 0,C 180,E1 19480.02,E2 19480.02} C_VEL
LIN {X 0,Y 480.926,Z 572.23,A -85,B 0,C 180,E1 19479.841,E2 19479.841} C_VEL
LIN {X 0,Y 470.994,Z 554.364,A -85,B 0,C 180,E1 19477.826,E2 19477.826} C_VEL
LIN {X 0,Y 460.328,Z 536.752,A -85,B 0,C 180,E1 19475.486,E2 19475.486} C_VEL
LIN {X 0,Y 448.855,Z 519.233,A -85,B 0,C 180,E1 19472.698,E2 19472.698} C_VEL
LIN {X 0,Y 442.183,Z 509.916,A -85,B 0,C 180,E1 19470.922,E2 19470.922} C_VEL
LIN {X 0,Y 436.194,Z 501.605,A -85,B 0,C 180,E1 19469.189,E2 19469.189} C_VEL
LIN {X 0,Y 432.346,Z 496.463,A -85,B 0,C 180,E1 19468.001,E2 19468.001} C_VEL
LIN {X 0,Y 425.315,Z 487.258,A -85,B 0,C 180,E1 19465.631,E2 19465.631} C_VEL
LIN {X 0,Y 421.448,Z 481.892,A -85,B 0,C 180,E1 19464.084,E2 19464.084} C_VEL
LIN {X 0,Y 418.669,Z 476.691,A -85,B 0,C 180,E1 19461.874,E2 19461.874} C_VEL
LIN {X 0,Y 416.571,Z 472.463,A -85,B 0,C 180,E1 19459.928,E2 19459.928} C_VEL
LIN {X 0,Y 414.666,Z 468.658,A -85,B 0,C 180,E1 19457.978,E2 19457.978} C_VEL
LIN {X 0,Y 411.401,Z 462.741,A -85,B 0,C 180,E1 19454.21,E2 19454.21} C_VEL
LIN {X 0,Y 408.732,Z 457.814,A -85,B 0,C 180,E1 19450.002,E2 19450.002} C_VEL
LIN {X 0,Y 406.344,Z 454.233,A -85,B 0,C 180,E1 19443.951,E2 19443.951} C_VEL
LIN {X 0,Y 406.121,Z 453.472,A -85,B 0,C 180,E1 19440.282,E2 19440.282} C_VEL
LIN {X 0,Y 406.337,Z 454.287,A -85,B 0,C 180,E1 19436.897,E2 19436.897} C_VEL
LIN {X 0,Y 408.501,Z 457.578,A -85,B 0,C 180,E1 19431.271,E2 19431.271} C_VEL
LIN {X 0,Y 409.28,Z 458.943,A -85,B 0,C 180,E1 19429.869,E2 19429.869} C_VEL
LIN {X 0,Y 412.108,Z 463.755,A -85,B 0,C 180,E1 19425.958,E2 19425.958} C_VEL
LIN {X 0,Y 414.261,Z 467.843,A -85,B 0,C 180,E1 19423.452,E2 19423.452} C_VEL
LIN {X 0,Y 415.313,Z 470,A -85,B 0,C 180,E1 19422.341,E2 19422.341} C_VEL
LIN {X 0,Y 420.097,Z 475.511,A -85,B 0,C 180,E1 19420.246,E2 19420.246} C_VEL
LIN {X 0,Y 425.52,Z 481.795,A -85,B 0,C 180,E1 19418.206,E2 19418.206} C_VEL
LIN {X 0,Y 430.443,Z 487.655,A -85,B 0,C 180,E1 19416.523,E2 19416.523} C_VEL
LIN {X 0,Y 434.484,Z 492.553,A -85,B 0,C 180,E1 19415.238,E2 19415.238} C_VEL
LIN {X 0,Y 438.9,Z 498.053,A -85,B 0,C 180,E1 19413.916,E2 19413.916} C_VEL
LIN {X 0,Y 445.993,Z 507.122,A -85,B 0,C 180,E1 19411.95,E2 19411.95} C_VEL
LIN {X 0,Y 455.777,Z 520.504,A -85,B 0,C 180,E1 19409.478,E2 19409.478} C_VEL
LIN {X 0,Y 467.282,Z 537.414,A -85,B 0,C 180,E1 19406.858,E2 19406.858} C_VEL
LIN {X 0,Y 478.916,Z 556.153,A -85,B 0,C 180,E1 19404.447,E2 19404.447} C_VEL
LIN {X 0,Y 483.029,Z 563.567,A -85,B 0,C 180,E1 19403.632,E2 19403.632} C_VEL
LIN {X 0,Y 470.93,Z 793.043,A -85,B 0,C 180,E1 19399.921,E2 19399.921} C_VEL
LIN {X 0,Y 467.945,Z 846.962,A -85,B 0,C 180,E1 19399.014,E2 19399.014} C_VEL
LIN {X 0,Y 465.4,Z 871.25,A -85,B 0,C 180,E1 19398.428,E2 19398.428} C_VEL
LIN {X 0,Y 462.317,Z 894.124,A -85,B 0,C 180,E1 19397.704,E2 19397.704} C_VEL
LIN {X 0,Y 458.43,Z 916.982,A -85,B 0,C 180,E1 19396.761,E2 19396.761} C_VEL
LIN {X 0,Y 454.483,Z 937.356,A -85,B 0,C 180,E1 19395.735,E2 19395.735} C_VEL
LIN {X 0,Y 449.311,Z 960.408,A -85,B 0,C 180,E1 19394.329,E2 19394.329} C_VEL
LIN {X 0,Y 444.646,Z 979.355,A -85,B 0,C 180,E1 19392.951,E2 19392.951} C_VEL
LIN {X 0,Y 438.833,Z 1000.915,A -85,B 0,C 180,E1 19391.099,E2 19391.099} C_VEL
LIN {X 0,Y 433.636,Z 1019.017,A -85,B 0,C 180,E1 19389.268,E2 19389.268} C_VEL
LIN {X 0,Y 427.654,Z 1038.906,A -85,B 0,C 180,E1 19386.905,E2 19386.905} C_VEL
LIN {X 0,Y 422.838,Z 1054.513,A -85,B 0,C 180,E1 19384.743,E2 19384.743} C_VEL
LIN {X 0,Y 417.475,Z 1071.744,A -85,B 0,C 180,E1 19381.959,E2 19381.959} C_VEL
LIN {X 0,Y 413.354,Z 1085.266,A -85,B 0,C 180,E1 19379.41,E2 19379.41} C_VEL
LIN {X 0,Y 409.173,Z 1099.572,A -85,B 0,C 180,E1 19376.251,E2 19376.251} C_VEL
LIN {X 0,Y 406.307,Z 1110.202,A -85,B 0,C 180,E1 19373.495,E2 19373.495} C_VEL
LIN {X 0,Y 403.577,Z 1121.601,A -85,B 0,C 180,E1 19369.993,E2 19369.993} C_VEL
LIN {X 0,Y 401.984,Z 1129.474,A -85,B 0,C 180,E1 19367.068,E2 19367.068} C_VEL
LIN {X 0,Y 400.822,Z 1136.936,A -85,B 0,C 180,E1 19363.709,E2 19363.709} C_VEL
LIN {X 0,Y 400.216,Z 1142.365,A -85,B 0,C 180,E1 19360.509,E2 19360.509} C_VEL
LIN {X 0,Y 399.976,Z 1146.258,A -85,B 0,C 180,E1 19357.469,E2 19357.469} C_VEL
LIN {X 0,Y 399.949,Z 1149.05,A -85,B 0,C 180,E1 19354.014,E2 19354.014} C_VEL
LIN {X 0,Y 399.953,Z 1150.079,A -85,B 0,C 180,E1 19351.146,E2 19351.146} C_VEL
LIN {X 0,Y 399.952,Z 1150.006,A -85,B 0,C 180,E1 19348.424,E2 19348.424} C_VEL
LIN {X 0,Y 399.933,Z 1148.542,A -85,B 0,C 180,E1 19345.124,E2 19345.124} C_VEL
LIN {X 0,Y 399.992,Z 1145.748,A -85,B 0,C 180,E1 19342.097,E2 19342.097} C_VEL
LIN {X 0,Y 400.256,Z 1141.922,A -85,B 0,C 180,E1 19339.201,E2 19339.201} C_VEL
LIN {X 0,Y 400.973,Z 1135.726,A -85,B 0,C 180,E1 19335.707,E2 19335.707} C_VEL
LIN {X 0,Y 402.113,Z 1128.716,A -85,B 0,C 180,E1 19332.639,E2 19332.639} C_VEL
LIN {X 0,Y 404.039,Z 1119.519,A -85,B 0,C 180,E1 19329.302,E2 19329.302} C_VEL
LIN {X 0,Y 406.609,Z 1108.969,A -85,B 0,C 180,E1 19326.176,E2 19326.176} C_VEL
LIN {X 0,Y 410.053,Z 1096.542,A -85,B 0,C 180,E1 19323.028,E2 19323.028} C_VEL
LIN {X 0,Y 413.982,Z 1083.05,A -85,B 0,C 180,E1 19320.162,E2 19320.162} C_VEL
LIN {X 0,Y 418.496,Z 1068.513,A -85,B 0,C 180,E1 19317.481,E2 19317.481} C_VEL
LIN {X 0,Y 423.542,Z 1052.058,A -85,B 0,C 180,E1 19314.911,E2 19314.911} C_VEL
LIN {X 0,Y 428.996,Z 1034.461,A -85,B 0,C 180,E1 19312.531,E2 19312.531} C_VEL
LIN {X 0,Y 434.522,Z 1015.79,A -85,B 0,C 180,E1 19310.401,E2 19310.401} C_VEL
LIN {X 0,Y 440.203,Z 995.934,A -85,B 0,C 180,E1 19308.451,E2 19308.451} C_VEL
LIN {X 0,Y 445.454,Z 975.874,A -85,B 0,C 180,E1 19306.794,E2 19306.794} C_VEL
LIN {X 0,Y 450.636,Z 954.701,A -85,B 0,C 180,E1 19305.301,E2 19305.301} C_VEL
LIN {X 0,Y 455.367,Z 932.526,A -85,B 0,C 180,E1 19304.018,E2 19304.018} C_VEL
LIN {X 0,Y 459.649,Z 910.042,A -85,B 0,C 180,E1 19302.936,E2 19302.936} C_VEL
LIN {X 0,Y 463.244,Z 886.964,A -85,B 0,C 180,E1 19302.066,E2 19302.066} C_VEL
LIN {X 0,Y 466.142,Z 864.59,A -85,B 0,C 180,E1 19301.401,E2 19301.401} C_VEL
LIN {X 0,Y 468.317,Z 839.93,A -85,B 0,C 180,E1 19300.868,E2 19300.868} C_VEL
LIN {X 0,Y 480.437,Z 609.562,A -85,B 0,C 180,E1 19297.117,E2 19297.117} C_VEL
LIN {X 0,Y 482.849,Z 562.986,A -85,B 0,C 180,E1 19296.354,E2 19296.354} C_VEL
LIN {X 0,Y 470.765,Z 542.94,A -85,B 0,C 180,E1 19293.923,E2 19293.923} C_VEL
LIN {X 0,Y 459.996,Z 526.693,A -85,B 0,C 180,E1 19291.559,E2 19291.559} C_VEL
LIN {X 0,Y 450.519,Z 513.282,A -85,B 0,C 180,E1 19289.276,E2 19289.276} C_VEL
LIN {X 0,Y 441.131,Z 500.813,A -85,B 0,C 180,E1 19286.776,E2 19286.776} C_VEL
LIN {X 0,Y 435.69,Z 494.092,A -85,B 0,C 180,E1 19285.196,E2 19285.196} C_VEL
LIN {X 0,Y 431.496,Z 488.9,A -85,B 0,C 180,E1 19283.888,E2 19283.888} C_VEL
LIN {X 0,Y 426.575,Z 483.038,A -85,B 0,C 180,E1 19282.244,E2 19282.244} C_VEL
LIN {X 0,Y 422.889,Z 478.768,A -85,B 0,C 180,E1 19280.918,E2 19280.918} C_VEL
LIN {X 0,Y 418.279,Z 473.501,A -85,B 0,C 180,E1 19279.117,E2 19279.117} C_VEL
LIN {X 0,Y 415.226,Z 469.78,A -85,B 0,C 180,E1 19277.663,E2 19277.663} C_VEL
LIN {X 0,Y 414.275,Z 467.871,A -85,B 0,C 180,E1 19276.692,E2 19276.692} C_VEL
LIN {X 0,Y 412.086,Z 463.747,A -85,B 0,C 180,E1 19274.186,E2 19274.186} C_VEL
LIN {X 0,Y 408.822,Z 457.866,A -85,B 0,C 180,E1 19269.431,E2 19269.431} C_VEL
LIN {X 0,Y 406.255,Z 454,A -85,B 0,C 180,E1 19263.245,E2 19263.245} C_VEL
LIN {X 0,Y 406.02,Z 453.093,A -85,B 0,C 180,E1 19259.718,E2 19259.718} C_VEL
LIN {X 0,Y 406.222,Z 453.852,A -85,B 0,C 180,E1 19256.048,E2 19256.048} C_VEL
LIN {X 0,Y 408.694,Z 457.75,A -85,B 0,C 180,E1 19249.712,E2 19249.712} C_VEL
LIN {X 0,Y 411.974,Z 463.78,A -85,B 0,C 180,E1 19244.804,E2 19244.804} C_VEL
LIN {X 0,Y 414.355,Z 468.011,A -85,B 0,C 180,E1 19242.153,E2 19242.153} C_VEL
LIN {X 0,Y 416.7,Z 472.593,A -85,B 0,C 180,E1 19239.785,E2 19239.785} C_VEL
LIN {X 0,Y 419.788,Z 478.849,A -85,B 0,C 180,E1 19237.006,E2 19237.006} C_VEL
LIN {X 0,Y 422.158,Z 483.151,A -85,B 0,C 180,E1 19235.363,E2 19235.363} C_VEL
LIN {X 0,Y 430.402,Z 494.001,A -85,B 0,C 180,E1 19232.464,E2 19232.464} C_VEL
LIN {X 0,Y 434.588,Z 499.467,A -85,B 0,C 180,E1 19231.145,E2 19231.145} C_VEL
LIN {X 0,Y 441.033,Z 508.348,A -85,B 0,C 180,E1 19229.253,E2 19229.253} C_VEL
LIN {X 0,Y 446.653,Z 516.237,A -85,B 0,C 180,E1 19227.73,E2 19227.73} C_VEL
LIN {X 0,Y 455.401,Z 529.263,A -85,B 0,C 180,E1 19225.533,E2 19225.533} C_VEL
LIN {X 0,Y 464.968,Z 544.33,A -85,B 0,C 180,E1 19223.341,E2 19223.341} C_VEL
LIN {X 0,Y 475.109,Z 561.71,A -85,B 0,C 180,E1 19221.198,E2 19221.198} C_VEL
LIN {X 0,Y 480.942,Z 572.612,A -85,B 0,C 180,E1 19220.03,E2 19220.03} C_VEL
LIN {X 0,Y 468.883,Z 826.951,A -85,B 0,C 180,E1 19216.119,E2 19216.119} C_VEL
LIN {X 0,Y 467.044,Z 855.647,A -85,B 0,C 180,E1 19215.615,E2 19215.615} C_VEL
LIN {X 0,Y 464.64,Z 877.979,A -85,B 0,C 180,E1 19215.062,E2 19215.062} C_VEL
LIN {X 0,Y 461.382,Z 900.505,A -85,B 0,C 180,E1 19214.297,E2 19214.297} C_VEL
LIN {X 0,Y 457.7,Z 921.557,A -85,B 0,C 180,E1 19213.393,E2 19213.393} C_VEL
LIN {X 0,Y 453.185,Z 943.139,A -85,B 0,C 180,E1 19212.232,E2 19212.232} C_VEL
LIN {X 0,Y 448.275,Z 963.908,A -85,B 0,C 180,E1 19210.886,E2 19210.886} C_VEL
LIN {X 0,Y 443.068,Z 983.296,A -85,B 0,C 180,E1 19209.357,E2 19209.357} C_VEL
LIN {X 0,Y 437.609,Z 1002.323,A -85,B 0,C 180,E1 19207.595,E2 19207.595} C_VEL
LIN {X 0,Y 432.141,Z 1019.733,A -85,B 0,C 180,E1 19205.668,E2 19205.668} C_VEL
LIN {X 0,Y 426.828,Z 1036.122,A -85,B 0,C 180,E1 19203.563,E2 19203.563} C_VEL
LIN {X 0,Y 421.742,Z 1051.096,A -85,B 0,C 180,E1 19201.28,E2 19201.28} C_VEL
LIN {X 0,Y 416.776,Z 1065.796,A -85,B 0,C 180,E1 19198.674,E2 19198.674} C_VEL
LIN {X 0,Y 412.521,Z 1078.336,A -85,B 0,C 180,E1 19196.022,E2 19196.022} C_VEL
LIN {X 0,Y 408.664,Z 1090.308,A -85,B 0,C 180,E1 19193.047,E2 19193.047} C_VEL
LIN {X 0,Y 405.691,Z 1100.097,A -85,B 0,C 180,E1 19190.109,E2 19190.109} C_VEL
LIN {X 0,Y 403.195,Z 1109.399,A -85,B 0,C 180,E1 19186.719,E2 19186.719} C_VEL
LIN {X 0,Y 401.688,Z 1116.068,A -85,B 0,C 180,E1 19183.679,E2 19183.679} C_VEL
LIN {X 0,Y 400.662,Z 1121.931,A -85,B 0,C 180,E1 19180.206,E2 19180.206} C_VEL
LIN {X 0,Y 400.197,Z 1125.617,A -85,B 0,C 180,E1 19177.176,E2 19177.176} C_VEL
LIN {X 0,Y 399.998,Z 1128.237,A -85,B 0,C 180,E1 19173.726,E2 19173.726} C_VEL
LIN {X 0,Y 399.968,Z 1129.149,A -85,B 0,C 180,E1 19170.859,E2 19170.859} C_VEL
LIN {X 0,Y 399.974,Z 1128.936,A -85,B 0,C 180,E1 19167.708,E2 19167.708} C_VEL
LIN {X 0,Y 400.066,Z 1127.198,A -85,B 0,C 180,E1 19164.55,E2 19164.55} C_VEL
LIN {X 0,Y 400.362,Z 1124.192,A -85,B 0,C 180,E1 19161.382,E2 19161.382} C_VEL
LIN {X 0,Y 400.541,Z 1122.704,A -85,B 0,C 180,E1 19160.252,E2 19160.252} C_VEL
LIN {X 0,Y 399.776,Z 1121.29,A -85,B 0,C 180,E1 19159.167,E2 19159.167} C_VEL
LIN {X 0,Y 394.353,Z 1116.74,A -85,B 0,C 180,E1 19156.185,E2 19156.185} C_VEL
LIN {X 0,Y 394.088,Z 1115.075,A -85,B 0,C 180,E1 19155.326,E2 19155.326} C_VEL
LIN {X 0,Y 396.047,Z 1107.352,A -85,B 0,C 180,E1 19151.908,E2 19151.908} C_VEL
LIN {X 0,Y 398.578,Z 1098.621,A -85,B 0,C 180,E1 19148.823,E2 19148.823} C_VEL
LIN {X 0,Y 402.349,Z 1087.001,A -85,B 0,C 180,E1 19145.445,E2 19145.445} C_VEL
LIN {X 0,Y 406.408,Z 1075.276,A -85,B 0,C 180,E1 19142.608,E2 19142.608} C_VEL
LIN {X 0,Y 411.305,Z 1061.347,A -85,B 0,C 180,E1 19139.786,E2 19139.786} C_VEL
LIN {X 0,Y 416.455,Z 1046.943,A -85,B 0,C 180,E1 19137.301,E2 19137.301} C_VEL
LIN {X 0,Y 421.913,Z 1031.116,A -85,B 0,C 180,E1 19135.004,E2 19135.004} C_VEL
LIN {X 0,Y 427.69,Z 1013.956,A -85,B 0,C 180,E1 19132.866,E2 19132.866} C_VEL
LIN {X 0,Y 433.396,Z 995.652,A -85,B 0,C 180,E1 19130.961,E2 19130.961} C_VEL
LIN {X 0,Y 439.001,Z 976.545,A -85,B 0,C 180,E1 19129.266,E2 19129.266} C_VEL
LIN {X 0,Y 444.047,Z 957.374,A -85,B 0,C 180,E1 19127.853,E2 19127.853} C_VEL
LIN {X 0,Y 449.14,Z 935.984,A -85,B 0,C 180,E1 19126.532,E2 19126.532} C_VEL
LIN {X 0,Y 453.176,Z 916.034,A -85,B 0,C 180,E1 19125.53,E2 19125.53} C_VEL
LIN {X 0,Y 457.061,Z 893.783,A -85,B 0,C 180,E1 19124.622,E2 19124.622} C_VEL
LIN {X 0,Y 460.012,Z 871.91,A -85,B 0,C 180,E1 19123.944,E2 19123.944} C_VEL
LIN {X 0,Y 462.408,Z 848.297,A -85,B 0,C 180,E1 19123.402,E2 19123.402} C_VEL
LIN {X 0,Y 465.932,Z 778.409,A -85,B 0,C 180,E1 19122.294,E2 19122.294} C_VEL
LIN {X 0,Y 475.942,Z 575.943,A -85,B 0,C 180,E1 19119.155,E2 19119.155} C_VEL
LIN {X 0,Y 466.472,Z 558.932,A -85,B 0,C 180,E1 19117.172,E2 19117.172} C_VEL
LIN {X 0,Y 456.838,Z 542.812,A -85,B 0,C 180,E1 19114.991,E2 19114.991} C_VEL
LIN {X 0,Y 445.888,Z 525.832,A -85,B 0,C 180,E1 19112.257,E2 19112.257} C_VEL
LIN {X 0,Y 439.221,Z 516.372,A -85,B 0,C 180,E1 19110.433,E2 19110.433} C_VEL
LIN {X 0,Y 433.441,Z 508.245,A -85,B 0,C 180,E1 19108.712,E2 19108.712} C_VEL
LIN {X 0,Y 429.758,Z 503.273,A -85,B 0,C 180,E1 19107.543,E2 19107.543} C_VEL
LIN {X 0,Y 423.128,Z 494.443,A -85,B 0,C 180,E1 19105.248,E2 19105.248} C_VEL
LIN {X 0,Y 418.763,Z 488.749,A -85,B 0,C 180,E1 19103.575,E2 19103.575} C_VEL
LIN {X 0,Y 412.761,Z 481.209,A -85,B 0,C 180,E1 19100.935,E2 19100.935} C_VEL
LIN {X 0,Y 411.702,Z 478.801,A -85,B 0,C 180,E1 19099.878,E2 19099.878} C_VEL
LIN {X 0,Y 409.696,Z 474.732,A -85,B 0,C 180,E1 19097.763,E2 19097.763} C_VEL
LIN {X 0,Y 406.587,Z 469.102,A -85,B 0,C 180,E1 19094.091,E2 19094.091} C_VEL
LIN {X 0,Y 403.965,Z 464.227,A -85,B 0,C 180,E1 19089.834,E2 19089.834} C_VEL
LIN {X 0,Y 401.727,Z 460.75,A -85,B 0,C 180,E1 19083.853,E2 19083.853} C_VEL
LIN {X 0,Y 401.532,Z 460.027,A -85,B 0,C 180,E1 19080.285,E2 19080.285} C_VEL
LIN {X 0,Y 401.745,Z 460.853,A -85,B 0,C 180,E1 19076.861,E2 19076.861} C_VEL
LIN {X 0,Y 404.044,Z 464.275,A -85,B 0,C 180,E1 19071.031,E2 19071.031} C_VEL
LIN {X 0,Y 404.769,Z 466.069,A -85,B 0,C 180,E1 19069.467,E2 19069.467} C_VEL
LIN {X 0,Y 407.307,Z 470.114,A -85,B 0,C 180,E1 19066.079,E2 19066.079} C_VEL
LIN {X 0,Y 408.471,Z 472.344,A -85,B 0,C 180,E1 19065.034,E2 19065.034} C_VEL
LIN {X 0,Y 412.979,Z 476.973,A -85,B 0,C 180,E1 19062.819,E2 19062.819} C_VEL
LIN {X 0,Y 418.779,Z 483.64,A -85,B 0,C 180,E1 19060.327,E2 19060.327} C_VEL
LIN {X 0,Y 423.998,Z 489.768,A -85,B 0,C 180,E1 19058.342,E2 19058.342} C_VEL
LIN {X 0,Y 431.268,Z 498.459,A -85,B 0,C 180,E1 19055.881,E2 19055.881} C_VEL
LIN {X 0,Y 439.559,Z 509.077,A -85,B 0,C 180,E1 19053.376,E2 19053.376} C_VEL
LIN {X 0,Y 450.18,Z 523.462,A -85,B 0,C 180,E1 19050.53,E2 19050.53} C_VEL
LIN {X 0,Y 459.555,Z 537.279,A -85,B 0,C 180,E1 19048.265,E2 19048.265} C_VEL
LIN {X 0,Y 469.012,Z 551.961,A -85,B 0,C 180,E1 19046.172,E2 19046.172} C_VEL
LIN {X 0,Y 477.914,Z 567.127,A -85,B 0,C 180,E1 19044.33,E2 19044.33} C_VEL
LIN {X 0,Y 465.503,Z 795.402,A -85,B 0,C 180,E1 19040.619,E2 19040.619} C_VEL
LIN {X 0,Y 462.548,Z 847.066,A -85,B 0,C 180,E1 19039.743,E2 19039.743} C_VEL
LIN {X 0,Y 459.94,Z 871.323,A -85,B 0,C 180,E1 19039.154,E2 19039.154} C_VEL
LIN {X 0,Y 456.77,Z 894.217,A -85,B 0,C 180,E1 19038.427,E2 19038.427} C_VEL
LIN {X 0,Y 452.65,Z 917.693,A -85,B 0,C 180,E1 19037.451,E2 19037.451} C_VEL
LIN {X 0,Y 448.361,Z 939.119,A -85,B 0,C 180,E1 19036.359,E2 19036.359} C_VEL
LIN {X 0,Y 443.271,Z 960.893,A -85,B 0,C 180,E1 19035.005,E2 19035.005} C_VEL
LIN {X 0,Y 438.465,Z 979.784,A -85,B 0,C 180,E1 19033.617,E2 19033.617} C_VEL
LIN {X 0,Y 432.466,Z 1001.251,A -85,B 0,C 180,E1 19031.75,E2 19031.75} C_VEL
LIN {X 0,Y 427.095,Z 1019.311,A -85,B 0,C 180,E1 19029.902,E2 19029.902} C_VEL
LIN {X 0,Y 420.952,Z 1038.956,A -85,B 0,C 180,E1 19027.537,E2 19027.537} C_VEL
LIN {X 0,Y 415.834,Z 1054.91,A -85,B 0,C 180,E1 19025.294,E2 19025.294} C_VEL
LIN {X 0,Y 410.405,Z 1071.641,A -85,B 0,C 180,E1 19022.544,E2 19022.544} C_VEL
LIN {X 0,Y 406.135,Z 1085.01,A -85,B 0,C 180,E1 19019.986,E2 19019.986} C_VEL
LIN {X 0,Y 401.75,Z 1099.329,A -85,B 0,C 180,E1 19016.775,E2 19016.775} C_VEL
LIN {X 0,Y 398.723,Z 1109.963,A -85,B 0,C 180,E1 19013.97,E2 19013.97} C_VEL
LIN {X 0,Y 395.829,Z 1121.372,A -85,B 0,C 180,E1 19010.402,E2 19010.402} C_VEL
LIN {X 0,Y 394.135,Z 1129.249,A -85,B 0,C 180,E1 19007.419,E2 19007.419} C_VEL
LIN {X 0,Y 392.894,Z 1136.717,A -85,B 0,C 180,E1 19003.991,E2 19003.991} C_VEL
LIN {X 0,Y 392.244,Z 1142.149,A -85,B 0,C 180,E1 19000.725,E2 19000.725} C_VEL
LIN {X 0,Y 391.978,Z 1146.044,A -85,B 0,C 180,E1 18997.623,E2 18997.623} C_VEL
LIN {X 0,Y 391.949,Z 1148.768,A -85,B 0,C 180,E1 18994.243,E2 18994.243} C_VEL
LIN {X 0,Y 391.956,Z 1149.846,A -85,B 0,C 180,E1 18991.316,E2 18991.316} C_VEL
LIN {X 0,Y 391.956,Z 1149.82,A -85,B 0,C 180,E1 18988.538,E2 18988.538} C_VEL
LIN {X 0,Y 391.935,Z 1148.448,A -85,B 0,C 180,E1 18985.171,E2 18985.171} C_VEL
LIN {X 0,Y 392.005,Z 1145.534,A -85,B 0,C 180,E1 18981.935,E2 18981.935} C_VEL
LIN {X 0,Y 392.286,Z 1141.704,A -85,B 0,C 180,E1 18978.979,E2 18978.979} C_VEL
LIN {X 0,Y 393.053,Z 1135.502,A -85,B 0,C 180,E1 18975.413,E2 18975.413} C_VEL
LIN {X 0,Y 394.274,Z 1128.488,A -85,B 0,C 180,E1 18972.282,E2 18972.282} C_VEL
LIN {X 0,Y 396.234,Z 1119.661,A -85,B 0,C 180,E1 18969.002,E2 18969.002} C_VEL
LIN {X 0,Y 399.001,Z 1108.865,A -85,B 0,C 180,E1 18965.733,E2 18965.733} C_VEL
LIN {X 0,Y 402.486,Z 1096.924,A -85,B 0,C 180,E1 18962.639,E2 18962.639} C_VEL
LIN {X 0,Y 406.678,Z 1083.167,A -85,B 0,C 180,E1 18959.655,E2 18959.655} C_VEL
LIN {X 0,Y 411.52,Z 1068.241,A -85,B 0,C 180,E1 18956.859,E2 18956.859} C_VEL
LIN {X 0,Y 416.78,Z 1051.771,A -85,B 0,C 180,E1 18954.255,E2 18954.255} C_VEL
LIN {X 0,Y 422.459,Z 1034.147,A -85,B 0,C 180,E1 18951.848,E2 18951.848} C_VEL
LIN {X 0,Y 428.011,Z 1016.078,A -85,B 0,C 180,E1 18949.763,E2 18949.763} C_VEL
LIN {X 0,Y 433.881,Z 996.305,A -85,B 0,C 180,E1 18947.796,E2 18947.796} C_VEL
LIN {X 0,Y 439.293,Z 976.294,A -85,B 0,C 180,E1 18946.125,E2 18946.125} C_VEL
LIN {X 0,Y 444.401,Z 956.122,A -85,B 0,C 180,E1 18944.684,E2 18944.684} C_VEL
LIN {X 0,Y 449.296,Z 934.123,A -85,B 0,C 180,E1 18943.384,E2 18943.384} C_VEL
LIN {X 0,Y 453.214,Z 914.306,A -85,B 0,C 180,E1 18942.406,E2 18942.406} C_VEL
LIN {X 0,Y 457.327,Z 889.729,A -85,B 0,C 180,E1 18941.432,E2 18941.432} C_VEL
LIN {X 0,Y 460.111,Z 869.247,A -85,B 0,C 180,E1 18940.8,E2 18940.8} C_VEL
LIN {X 0,Y 462.683,Z 843.641,A -85,B 0,C 180,E1 18940.205,E2 18940.205} C_VEL
LIN {X 0,Y 470.36,Z 702.745,A -85,B 0,C 180,E1 18937.88,E2 18937.88} C_VEL
LIN {X 0,Y 477.741,Z 566.721,A -85,B 0,C 180,E1 18935.662,E2 18935.662} C_VEL
LIN {X 0,Y 465.853,Z 546.978,A -85,B 0,C 180,E1 18933.184,E2 18933.184} C_VEL
LIN {X 0,Y 454.608,Z 529.901,A -85,B 0,C 180,E1 18930.609,E2 18930.609} C_VEL
LIN {X 0,Y 445.467,Z 517.128,A -85,B 0,C 180,E1 18928.305,E2 18928.305} C_VEL
LIN {X 0,Y 437.623,Z 506.718,A -85,B 0,C 180,E1 18926.13,E2 18926.13} C_VEL
LIN {X 0,Y 433.009,Z 500.857,A -85,B 0,C 180,E1 18924.742,E2 18924.742} C_VEL
LIN {X 0,Y 428.981,Z 495.814,A -85,B 0,C 180,E1 18923.453,E2 18923.453} C_VEL
LIN {X 0,Y 423.278,Z 488.918,A -85,B 0,C 180,E1 18921.478,E2 18921.478} C_VEL
LIN {X 0,Y 416.663,Z 481.181,A -85,B 0,C 180,E1 18918.903,E2 18918.903} C_VEL
LIN {X 0,Y 411.33,Z 475.215,A -85,B 0,C 180,E1 18916.524,E2 18916.524} C_VEL
LIN {X 0,Y 407.586,Z 470.959,A -85,B 0,C 180,E1 18914.491,E2 18914.491} C_VEL
LIN {X 0,Y 406.836,Z 469.303,A -85,B 0,C 180,E1 18913.502,E2 18913.502} C_VEL
LIN {X 0,Y 404.068,Z 464.28,A -85,B 0,C 180,E1 18909.256,E2 18909.256} C_VEL
LIN {X 0,Y 401.646,Z 460.514,A -85,B 0,C 180,E1 18903.14,E2 18903.14} C_VEL
LIN {X 0,Y 401.432,Z 459.648,A -85,B 0,C 180,E1 18899.715,E2 18899.715} C_VEL
LIN {X 0,Y 401.607,Z 460.369,A -85,B 0,C 180,E1 18896.145,E2 18896.145} C_VEL
LIN {X 0,Y 403.822,Z 464.067,A -85,B 0,C 180,E1 18890.019,E2 18890.019} C_VEL
LIN {X 0,Y 404.477,Z 465.403,A -85,B 0,C 180,E1 18888.738,E2 18888.738} C_VEL
LIN {X 0,Y 407.151,Z 470.133,A -85,B 0,C 180,E1 18884.911,E2 18884.911} C_VEL
LIN {X 0,Y 409.511,Z 474.361,A -85,B 0,C 180,E1 18882.224,E2 18882.224} C_VEL
LIN {X 0,Y 411.644,Z 478.711,A -85,B 0,C 180,E1 18879.971,E2 18879.971} C_VEL
LIN {X 0,Y 413.548,Z 482.375,A -85,B 0,C 180,E1 18878.438,E2 18878.438} C_VEL
LIN {X 0,Y 417.058,Z 486.862,A -85,B 0,C 180,E1 18876.922,E2 18876.922} C_VEL
LIN {X 0,Y 420.258,Z 490.7,A -85,B 0,C 180,E1 18875.657,E2 18875.657} C_VEL
LIN {X 0,Y 427.942,Z 500.895,A -85,B 0,C 180,E1 18872.895,E2 18872.895} C_VEL
LIN {X 0,Y 432.344,Z 506.792,A -85,B 0,C 180,E1 18871.473,E2 18871.473} C_VEL
LIN {X 0,Y 438.294,Z 515.093,A -85,B 0,C 180,E1 18869.686,E2 18869.686} C_VEL
LIN {X 0,Y 444.034,Z 523.304,A -85,B 0,C 180,E1 18868.09,E2 18868.09} C_VEL
LIN {X 0,Y 453.963,Z 538.315,A -85,B 0,C 180,E1 18865.562,E2 18865.562} C_VEL
LIN {X 0,Y 463.962,Z 554.685,A -85,B 0,C 180,E1 18863.251,E2 18863.251} C_VEL
LIN {X 0,Y 473.789,Z 572.057,A -85,B 0,C 180,E1 18861.16,E2 18861.16} C_VEL
LIN {X 0,Y 475.842,Z 576.277,A -85,B 0,C 180,E1 18860.733,E2 18860.733} C_VEL
LIN {X 0,Y 463.433,Z 829.177,A -85,B 0,C 180,E1 18856.819,E2 18856.819} C_VEL
LIN {X 0,Y 461.596,Z 856.124,A -85,B 0,C 180,E1 18856.336,E2 18856.336} C_VEL
LIN {X 0,Y 459.044,Z 879.069,A -85,B 0,C 180,E1 18855.76,E2 18855.76} C_VEL
LIN {X 0,Y 455.586,Z 901.92,A -85,B 0,C 180,E1 18854.968,E2 18854.968} C_VEL
LIN {X 0,Y 451.71,Z 923.334,A -85,B 0,C 180,E1 18854.032,E2 18854.032} C_VEL
LIN {X 0,Y 446.993,Z 944.871,A -85,B 0,C 180,E1 18852.846,E2 18852.846} C_VEL
LIN {X 0,Y 441.809,Z 965.866,A -85,B 0,C 180,E1 18851.451,E2 18851.451} C_VEL
LIN {X 0,Y 436.659,Z 984.386,A -85,B 0,C 180,E1 18849.964,E2 18849.964} C_VEL
LIN {X 0,Y 430.838,Z 1003.844,A -85,B 0,C 180,E1 18848.122,E2 18848.122} C_VEL
LIN {X 0,Y 425.405,Z 1020.583,A -85,B 0,C 180,E1 18846.238,E2 18846.238} C_VEL
LIN {X 0,Y 419.575,Z 1037.793,A -85,B 0,C 180,E1 18843.971,E2 18843.971} C_VEL
LIN {X 0,Y 414.514,Z 1052.193,A -85,B 0,C 180,E1 18841.726,E2 18841.726} C_VEL
LIN {X 0,Y 409.13,Z 1067.417,A -85,B 0,C 180,E1 18838.941,E2 18838.941} C_VEL
LIN {X 0,Y 404.781,Z 1079.822,A -85,B 0,C 180,E1 18836.242,E2 18836.242} C_VEL
LIN {X 0,Y 400.654,Z 1092.046,A -85,B 0,C 180,E1 18833.068,E2 18833.068} C_VEL
LIN {X 0,Y 397.592,Z 1101.885,A -85,B 0,C 180,E1 18830,E2 18830} C_VEL
LIN {X 0,Y 395.225,Z 1110.306,A -85,B 0,C 180,E1 18826.763,E2 18826.763} C_VEL
LIN {X 0,Y 393.637,Z 1117.168,A -85,B 0,C 180,E1 18823.515,E2 18823.515} C_VEL
LIN {X 0,Y 392.648,Z 1122.544,A -85,B 0,C 180,E1 18820.12,E2 18820.12} C_VEL
LIN {X 0,Y 392.18,Z 1126.292,A -85,B 0,C 180,E1 18816.882,E2 18816.882} C_VEL
LIN {X 0,Y 391.996,Z 1128.578,A -85,B 0,C 180,E1 18813.51,E2 18813.51} C_VEL
LIN {X 0,Y 391.968,Z 1129.402,A -85,B 0,C 180,E1 18810.585,E2 18810.585} C_VEL
LIN {X 0,Y 391.98,Z 1128.951,A -85,B 0,C 180,E1 18807.222,E2 18807.222} C_VEL
LIN {X 0,Y 392.086,Z 1127.3,A -85,B 0,C 180,E1 18804.292,E2 18804.292} C_VEL
LIN {X 0,Y 392.456,Z 1124.077,A -85,B 0,C 180,E1 18800.911,E2 18800.911} C_VEL
LIN {X 0,Y 393.238,Z 1119.111,A -85,B 0,C 180,E1 18797.518,E2 18797.518} C_VEL
LIN {X 0,Y 394.088,Z 1115.075,A -85,B 0,C 180,E1 18795.326,E2 18795.326} C_VEL
LIN {X 0,Y 393.633,Z 1112.999,A -85,B 0,C 180,E1 18794.243,E2 18794.243} C_VEL
LIN {X 0,Y 389.204,Z 1106.938,A -85,B 0,C 180,E1 18791.329,E2 18791.329} C_VEL
LIN {X 0,Y 389.166,Z 1104.616,A -85,B 0,C 180,E1 18790.405,E2 18790.405} C_VEL
LIN {X 0,Y 392.555,Z 1094.117,A -85,B 0,C 180,E1 18786.905,E2 18786.905} C_VEL
LIN {X 0,Y 396.386,Z 1083.216,A -85,B 0,C 180,E1 18783.899,E2 18783.899} C_VEL
LIN {X 0,Y 401.109,Z 1070.179,A -85,B 0,C 180,E1 18780.915,E2 18780.915} C_VEL
LIN {X 0,Y 406.298,Z 1056.31,A -85,B 0,C 180,E1 18778.22,E2 18778.22} C_VEL
LIN {X 0,Y 411.87,Z 1040.91,A -85,B 0,C 180,E1 18775.721,E2 18775.721} C_VEL
LIN {X 0,Y 417.803,Z 1024.331,A -85,B 0,C 180,E1 18773.422,E2 18773.422} C_VEL
LIN {X 0,Y 423.516,Z 1007.343,A -85,B 0,C 180,E1 18771.443,E2 18771.443} C_VEL
LIN {X 0,Y 429.482,Z 988.59,A -85,B 0,C 180,E1 18769.579,E2 18769.579} C_VEL
LIN {X 0,Y 434.705,Z 970.5,A -85,B 0,C 180,E1 18768.072,E2 18768.072} C_VEL
LIN {X 0,Y 440.144,Z 950.053,A -85,B 0,C 180,E1 18766.632,E2 18766.632} C_VEL
LIN {X 0,Y 444.915,Z 929.222,A -85,B 0,C 180,E1 18765.432,E2 18765.432} C_VEL
LIN {X 0,Y 449.273,Z 907.414,A -85,B 0,C 180,E1 18764.405,E2 18764.405} C_VEL
LIN {X 0,Y 452.788,Z 885.667,A -85,B 0,C 180,E1 18763.604,E2 18763.604} C_VEL
LIN {X 0,Y 455.8,Z 862.025,A -85,B 0,C 180,E1 18762.944,E2 18762.944} C_VEL
LIN {X 0,Y 457.664,Z 839.848,A -85,B 0,C 180,E1 18762.504,E2 18762.504} C_VEL
LIN {X 0,Y 470.486,Z 588.385,A -85,B 0,C 180,E1 18758.578,E2 18758.578} C_VEL
LIN {X 0,Y 470.83,Z 579.38,A -85,B 0,C 180,E1 18758.416,E2 18758.416} C_VEL
LIN {X 0,Y 460.872,Z 561.35,A -85,B 0,C 180,E1 18756.243,E2 18756.243} C_VEL
LIN {X 0,Y 451.532,Z 545.903,A -85,B 0,C 180,E1 18754.035,E2 18754.035} C_VEL
LIN {X 0,Y 442.509,Z 531.83,A -85,B 0,C 180,E1 18751.692,E2 18751.692} C_VEL
LIN {X 0,Y 436.19,Z 522.671,A -85,B 0,C 180,E1 18749.906,E2 18749.906} C_VEL
LIN {X 0,Y 428.532,Z 511.67,A -85,B 0,C 180,E1 18747.516,E2 18747.516} C_VEL
LIN {X 0,Y 420.442,Z 501.021,A -85,B 0,C 180,E1 18744.669,E2 18744.669} C_VEL
LIN {X 0,Y 416.674,Z 495.966,A -85,B 0,C 180,E1 18743.176,E2 18743.176} C_VEL
LIN {X 0,Y 409.32,Z 486.497,A -85,B 0,C 180,E1 18739.85,E2 18739.85} C_VEL
LIN {X 0,Y 405.704,Z 482.231,A -85,B 0,C 180,E1 18737.943,E2 18737.943} C_VEL
LIN {X 0,Y 404.402,Z 480.363,A -85,B 0,C 180,E1 18737.111,E2 18737.111} C_VEL
LIN {X 0,Y 401.912,Z 475.607,A -85,B 0,C 180,E1 18734.111,E2 18734.111} C_VEL
LIN {X 0,Y 399.303,Z 470.726,A -85,B 0,C 180,E1 18729.804,E2 18729.804} C_VEL
LIN {X 0,Y 397.113,Z 467.267,A -85,B 0,C 180,E1 18723.754,E2 18723.754} C_VEL
LIN {X 0,Y 396.951,Z 466.572,A -85,B 0,C 180,E1 18720.144,E2 18720.144} C_VEL
LIN {X 0,Y 397.215,Z 467.532,A -85,B 0,C 180,E1 18716.536,E2 18716.536} C_VEL
LIN {X 0,Y 399.69,Z 471.087,A -85,B 0,C 180,E1 18710.642,E2 18710.642} C_VEL
LIN {X 0,Y 400.634,Z 473.236,A -85,B 0,C 180,E1 18709.212,E2 18709.212} C_VEL
LIN {X 0,Y 405.4,Z 477.981,A -85,B 0,C 180,E1 18706.158,E2 18706.158} C_VEL
LIN {X 0,Y 410.169,Z 483.204,A -85,B 0,C 180,E1 18703.647,E2 18703.647} C_VEL
LIN {X 0,Y 416.985,Z 491.18,A -85,B 0,C 180,E1 18700.603,E2 18700.603} C_VEL
LIN {X 0,Y 422.656,Z 497.941,A -85,B 0,C 180,E1 18698.415,E2 18698.415} C_VEL
LIN {X 0,Y 429.773,Z 506.808,A -85,B 0,C 180,E1 18695.974,E2 18695.974} C_VEL
LIN {X 0,Y 436.797,Z 515.786,A -85,B 0,C 180,E1 18693.817,E2 18693.817} C_VEL
LIN {X 0,Y 447.477,Z 530.489,A -85,B 0,C 180,E1 18690.885,E2 18690.885} C_VEL
LIN {X 0,Y 458.046,Z 546.263,A -85,B 0,C 180,E1 18688.295,E2 18688.295} C_VEL
LIN {X 0,Y 467.495,Z 561.588,A -85,B 0,C 180,E1 18686.177,E2 18686.177} C_VEL
LIN {X 0,Y 472.854,Z 570.999,A -85,B 0,C 180,E1 18685.039,E2 18685.039} C_VEL
LIN {X 0,Y 460.128,Z 798.203,A -85,B 0,C 180,E1 18681.326,E2 18681.326} C_VEL
LIN {X 0,Y 457.201,Z 847.488,A -85,B 0,C 180,E1 18680.483,E2 18680.483} C_VEL
LIN {X 0,Y 454.534,Z 871.569,A -85,B 0,C 180,E1 18679.894,E2 18679.894} C_VEL
LIN {X 0,Y 451.297,Z 894.316,A -85,B 0,C 180,E1 18679.168,E2 18679.168} C_VEL
LIN {X 0,Y 447.179,Z 917.179,A -85,B 0,C 180,E1 18678.216,E2 18678.216} C_VEL
LIN {X 0,Y 443.006,Z 937.465,A -85,B 0,C 180,E1 18677.185,E2 18677.185} C_VEL
LIN {X 0,Y 437.53,Z 960.471,A -85,B 0,C 180,E1 18675.762,E2 18675.762} C_VEL
LIN {X 0,Y 432.562,Z 979.394,A -85,B 0,C 180,E1 18674.367,E2 18674.367} C_VEL
LIN {X 0,Y 426.366,Z 1000.911,A -85,B 0,C 180,E1 18672.486,E2 18672.486} C_VEL
LIN {X 0,Y 420.992,Z 1018.372,A -85,B 0,C 180,E1 18670.69,E2 18670.69} C_VEL
LIN {X 0,Y 414.587,Z 1038.147,A -85,B 0,C 180,E1 18668.304,E2 18668.304} C_VEL
LIN {X 0,Y 409.308,Z 1053.949,A -85,B 0,C 180,E1 18666.067,E2 18666.067} C_VEL
LIN {X 0,Y 403.492,Z 1071.22,A -85,B 0,C 180,E1 18663.207,E2 18663.207} C_VEL
LIN {X 0,Y 398.961,Z 1084.755,A -85,B 0,C 180,E1 18660.582,E2 18660.582} C_VEL
LIN {X 0,Y 394.363,Z 1099.087,A -85,B 0,C 180,E1 18657.317,E2 18657.317} C_VEL
LIN {X 0,Y 391.162,Z 1109.726,A -85,B 0,C 180,E1 18654.463,E2 18654.463} C_VEL
LIN {X 0,Y 388.203,Z 1120.725,A -85,B 0,C 180,E1 18650.979,E2 18650.979} C_VEL
LIN {X 0,Y 386.373,Z 1128.659,A -85,B 0,C 180,E1 18647.936,E2 18647.936} C_VEL
LIN {X 0,Y 385.01,Z 1136.232,A -85,B 0,C 180,E1 18644.437,E2 18644.437} C_VEL
LIN {X 0,Y 384.274,Z 1141.933,A -85,B 0,C 180,E1 18640.95,E2 18640.95} C_VEL
LIN {X 0,Y 383.993,Z 1145.665,A -85,B 0,C 180,E1 18637.933,E2 18637.933} C_VEL
LIN {X 0,Y 383.947,Z 1148.486,A -85,B 0,C 180,E1 18634.481,E2 18634.481} C_VEL
LIN {X 0,Y 383.959,Z 1149.636,A -85,B 0,C 180,E1 18631.343,E2 18631.343} C_VEL
LIN {X 0,Y 383.958,Z 1149.61,A -85,B 0,C 180,E1 18628.508,E2 18628.508} C_VEL
LIN {X 0,Y 383.937,Z 1148.336,A -85,B 0,C 180,E1 18625.22,E2 18625.22} C_VEL
LIN {X 0,Y 384.006,Z 1145.486,A -85,B 0,C 180,E1 18621.917,E2 18621.917} C_VEL
LIN {X 0,Y 384.296,Z 1141.702,A -85,B 0,C 180,E1 18618.899,E2 18618.899} C_VEL
LIN {X 0,Y 385.052,Z 1135.906,A -85,B 0,C 180,E1 18615.411,E2 18615.411} C_VEL
LIN {X 0,Y 386.371,Z 1128.626,A -85,B 0,C 180,E1 18612.064,E2 18612.064} C_VEL
LIN {X 0,Y 388.42,Z 1119.854,A -85,B 0,C 180,E1 18608.717,E2 18608.717} C_VEL
LIN {X 0,Y 391.307,Z 1109.153,A -85,B 0,C 180,E1 18605.386,E2 18605.386} C_VEL
LIN {X 0,Y 394.74,Z 1097.858,A -85,B 0,C 180,E1 18602.384,E2 18602.384} C_VEL
LIN {X 0,Y 399.183,Z 1083.966,A -85,B 0,C 180,E1 18599.27,E2 18599.27} C_VEL
LIN {X 0,Y 403.758,Z 1070.349,A -85,B 0,C 180,E1 18596.648,E2 18596.648} C_VEL
LIN {X 0,Y 409.45,Z 1053.374,A -85,B 0,C 180,E1 18593.86,E2 18593.86} C_VEL
LIN {X 0,Y 414.746,Z 1037.514,A -85,B 0,C 180,E1 18591.626,E2 18591.626} C_VEL
LIN {X 0,Y 420.974,Z 1018.222,A -85,B 0,C 180,E1 18589.308,E2 18589.308} C_VEL
LIN {X 0,Y 426.347,Z 1000.738,A -85,B 0,C 180,E1 18587.512,E2 18587.512} C_VEL
LIN {X 0,Y 432.539,Z 979.18,A -85,B 0,C 180,E1 18585.63,E2 18585.63} C_VEL
LIN {X 0,Y 437.273,Z 961.148,A -85,B 0,C 180,E1 18584.297,E2 18584.297} C_VEL
LIN {X 0,Y 442.505,Z 939.449,A -85,B 0,C 180,E1 18582.936,E2 18582.936} C_VEL
LIN {X 0,Y 446.912,Z 918.066,A -85,B 0,C 180,E1 18581.838,E2 18581.838} C_VEL
LIN {X 0,Y 451.006,Z 895.471,A -85,B 0,C 180,E1 18580.886,E2 18580.886} C_VEL
LIN {X 0,Y 454.378,Z 871.992,A -85,B 0,C 180,E1 18580.129,E2 18580.129} C_VEL
LIN {X 0,Y 457.031,Z 848.159,A -85,B 0,C 180,E1 18579.544,E2 18579.544} C_VEL
LIN {X 0,Y 459.669,Z 804.775,A -85,B 0,C 180,E1 18578.793,E2 18578.793} C_VEL
LIN {X 0,Y 472.332,Z 577.974,A -85,B 0,C 180,E1 18575.085,E2 18575.085} C_VEL
LIN {X 0,Y 472.649,Z 570.441,A -85,B 0,C 180,E1 18574.944,E2 18574.944} C_VEL
LIN {X 0,Y 461.863,Z 552.396,A -85,B 0,C 180,E1 18572.62,E2 18572.62} C_VEL
LIN {X 0,Y 450.923,Z 535.639,A -85,B 0,C 180,E1 18570.039,E2 18570.039} C_VEL
LIN {X 0,Y 442.497,Z 523.705,A -85,B 0,C 180,E1 18567.852,E2 18567.852} C_VEL
LIN {X 0,Y 434.785,Z 513.331,A -85,B 0,C 180,E1 18565.653,E2 18565.653} C_VEL
LIN {X 0,Y 427.807,Z 504.22,A -85,B 0,C 180,E1 18563.448,E2 18563.448} C_VEL
LIN {X 0,Y 419.561,Z 494.18,A -85,B 0,C 180,E1 18560.507,E2 18560.507} C_VEL
LIN {X 0,Y 414.423,Z 488.28,A -85,B 0,C 180,E1 18558.425,E2 18558.425} C_VEL
LIN {X 0,Y 409.791,Z 482.896,A -85,B 0,C 180,E1 18556.296,E2 18556.296} C_VEL
LIN {X 0,Y 404.205,Z 476.756,A -85,B 0,C 180,E1 18553.3,E2 18553.3} C_VEL
LIN {X 0,Y 400.011,Z 472.18,A -85,B 0,C 180,E1 18550.368,E2 18550.368} C_VEL
LIN {X 0,Y 399.314,Z 470.689,A -85,B 0,C 180,E1 18549.077,E2 18549.077} C_VEL
LIN {X 0,Y 397.03,Z 467.022,A -85,B 0,C 180,E1 18543.032,E2 18543.032} C_VEL
LIN {X 0,Y 396.83,Z 466.214,A -85,B 0,C 180,E1 18539.567,E2 18539.567} C_VEL
LIN {X 0,Y 397.033,Z 466.988,A -85,B 0,C 180,E1 18535.956,E2 18535.956} C_VEL
LIN {X 0,Y 399.54,Z 470.992,A -85,B 0,C 180,E1 18529.473,E2 18529.473} C_VEL
LIN {X 0,Y 402.332,Z 476.487,A -85,B 0,C 180,E1 18525.021,E2 18525.021} C_VEL
LIN {X 0,Y 404.672,Z 480.652,A -85,B 0,C 180,E1 18522.455,E2 18522.455} C_VEL
LIN {X 0,Y 408.64,Z 485.889,A -85,B 0,C 180,E1 18520.265,E2 18520.265} C_VEL
LIN {X 0,Y 414.391,Z 493.196,A -85,B 0,C 180,E1 18517.589,E2 18517.589} C_VEL
LIN {X 0,Y 418.299,Z 498.113,A -85,B 0,C 180,E1 18515.986,E2 18515.986} C_VEL
LIN {X 0,Y 425.597,Z 507.926,A -85,B 0,C 180,E1 18513.3,E2 18513.3} C_VEL
LIN {X 0,Y 430.21,Z 514.246,A -85,B 0,C 180,E1 18511.772,E2 18511.772} C_VEL
LIN {X 0,Y 435.884,Z 522.301,A -85,B 0,C 180,E1 18510.033,E2 18510.033} C_VEL
LIN {X 0,Y 441.554,Z 530.543,A -85,B 0,C 180,E1 18508.422,E2 18508.422} C_VEL
LIN {X 0,Y 450.896,Z 544.932,A -85,B 0,C 180,E1 18505.987,E2 18505.987} C_VEL
LIN {X 0,Y 460.64,Z 561.105,A -85,B 0,C 180,E1 18503.678,E2 18503.678} C_VEL
LIN {X 0,Y 470.44,Z 578.802,A -85,B 0,C 180,E1 18501.541,E2 18501.541} C_VEL
LIN {X 0,Y 470.806,Z 580.08,A -85,B 0,C 180,E1 18501.45,E2 18501.45} C_VEL
LIN {X 0,Y 458.06,Z 831.261,A -85,B 0,C 180,E1 18497.537,E2 18497.537} C_VEL
LIN {X 0,Y 456.223,Z 856.597,A -85,B 0,C 180,E1 18497.073,E2 18497.073} C_VEL
LIN {X 0,Y 453.531,Z 879.988,A -85,B 0,C 180,E1 18496.48,E2 18496.48} C_VEL
LIN {X 0,Y 449.981,Z 902.593,A -85,B 0,C 180,E1 18495.685,E2 18495.685} C_VEL
LIN {X 0,Y 445.747,Z 924.995,A -85,B 0,C 180,E1 18494.688,E2 18494.688} C_VEL
LIN {X 0,Y 441.152,Z 945.336,A -85,B 0,C 180,E1 18493.554,E2 18493.554} C_VEL
LIN {X 0,Y 435.816,Z 966.255,A -85,B 0,C 180,E1 18492.151,E2 18492.151} C_VEL
LIN {X 0,Y 430.511,Z 984.748,A -85,B 0,C 180,E1 18490.653,E2 18490.653} C_VEL
LIN {X 0,Y 424.506,Z 1004.162,A -85,B 0,C 180,E1 18488.796,E2 18488.796} C_VEL
LIN {X 0,Y 418.963,Z 1020.692,A -85,B 0,C 180,E1 18486.917,E2 18486.917} C_VEL
LIN {X 0,Y 413.044,Z 1037.585,A -85,B 0,C 180,E1 18484.673,E2 18484.673} C_VEL
LIN {X 0,Y 407.608,Z 1052.46,A -85,B 0,C 180,E1 18482.328,E2 18482.328} C_VEL
LIN {X 0,Y 402.014,Z 1067.668,A -85,B 0,C 180,E1 18479.503,E2 18479.503} C_VEL
LIN {X 0,Y 397.42,Z 1080.223,A -85,B 0,C 180,E1 18476.726,E2 18476.726} C_VEL
LIN {X 0,Y 393.156,Z 1092.28,A -85,B 0,C 180,E1 18473.534,E2 18473.534} C_VEL
LIN {X 0,Y 389.941,Z 1102.116,A -85,B 0,C 180,E1 18470.41,E2 18470.41} C_VEL
LIN {X 0,Y 387.442,Z 1110.529,A -85,B 0,C 180,E1 18467.11,E2 18467.11} C_VEL
LIN {X 0,Y 385.698,Z 1117.677,A -85,B 0,C 180,E1 18463.645,E2 18463.645} C_VEL
LIN {X 0,Y 384.67,Z 1122.958,A -85,B 0,C 180,E1 18460.181,E2 18460.181} C_VEL
LIN {X 0,Y 384.174,Z 1126.781,A -85,B 0,C 180,E1 18456.726,E2 18456.726} C_VEL
LIN {X 0,Y 383.998,Z 1128.854,A -85,B 0,C 180,E1 18453.433,E2 18453.433} C_VEL
LIN {X 0,Y 383.971,Z 1129.656,A -85,B 0,C 180,E1 18450.298,E2 18450.298} C_VEL
LIN {X 0,Y 383.992,Z 1129.03,A -85,B 0,C 180,E1 18446.865,E2 18446.865} C_VEL
LIN {X 0,Y 384.117,Z 1127.293,A -85,B 0,C 180,E1 18443.873,E2 18443.873} C_VEL
LIN {X 0,Y 384.555,Z 1123.694,A -85,B 0,C 180,E1 18440.27,E2 18440.27} C_VEL
LIN {X 0,Y 385.384,Z 1119.081,A -85,B 0,C 180,E1 18437.107,E2 18437.107} C_VEL
LIN {X 0,Y 387.077,Z 1111.949,A -85,B 0,C 180,E1 18433.409,E2 18433.409} C_VEL
LIN {X 0,Y 389.166,Z 1104.616,A -85,B 0,C 180,E1 18430.405,E2 18430.405} C_VEL
LIN {X 0,Y 389.086,Z 1101.871,A -85,B 0,C 180,E1 18429.336,E2 18429.336} C_VEL
LIN {X 0,Y 385.855,Z 1094.685,A -85,B 0,C 180,E1 18426.595,E2 18426.595} C_VEL
LIN {X 0,Y 386.118,Z 1091.414,A -85,B 0,C 180,E1 18425.547,E2 18425.547} C_VEL
LIN {X 0,Y 390.646,Z 1079.205,A -85,B 0,C 180,E1 18422.328,E2 18422.328} C_VEL
LIN {X 0,Y 395.623,Z 1066.311,A -85,B 0,C 180,E1 18419.469,E2 18419.469} C_VEL
LIN {X 0,Y 401.229,Z 1051.609,A -85,B 0,C 180,E1 18416.752,E2 18416.752} C_VEL
LIN {X 0,Y 407.293,Z 1035.666,A -85,B 0,C 180,E1 18414.247,E2 18414.247} C_VEL
LIN {X 0,Y 413.227,Z 1019.16,A -85,B 0,C 180,E1 18412.076,E2 18412.076} C_VEL
LIN {X 0,Y 419.524,Z 1000.855,A -85,B 0,C 180,E1 18410.025,E2 18410.025} C_VEL
LIN {X 0,Y 425.338,Z 982.409,A -85,B 0,C 180,E1 18408.296,E2 18408.296} C_VEL
LIN {X 0,Y 431.327,Z 961.764,A -85,B 0,C 180,E1 18406.671,E2 18406.671} C_VEL
LIN {X 0,Y 436.395,Z 942.067,A -85,B 0,C 180,E1 18405.39,E2 18405.39} C_VEL
LIN {X 0,Y 441.406,Z 919.726,A -85,B 0,C 180,E1 18404.197,E2 18404.197} C_VEL
LIN {X 0,Y 445.28,Z 899.203,A -85,B 0,C 180,E1 18403.318,E2 18403.318} C_VEL
LIN {X 0,Y 448.982,Z 874.819,A -85,B 0,C 180,E1 18402.511,E2 18402.511} C_VEL
LIN {X 0,Y 451.461,Z 852.942,A -85,B 0,C 180,E1 18401.98,E2 18401.98} C_VEL
LIN {X 0,Y 453.529,Z 820.429,A -85,B 0,C 180,E1 18401.423,E2 18401.423} C_VEL
LIN {X 0,Y 465.991,Z 583.113,A -85,B 0,C 180,E1 18397.701,E2 18397.701} C_VEL
LIN {X 0,Y 456.38,Z 565.736,A -85,B 0,C 180,E1 18395.531,E2 18395.531} C_VEL
LIN {X 0,Y 447.255,Z 550.423,A -85,B 0,C 180,E1 18393.288,E2 18393.288} C_VEL
LIN {X 0,Y 437.606,Z 535.368,A -85,B 0,C 180,E1 18390.671,E2 18390.671} C_VEL
LIN {X 0,Y 429.175,Z 523.075,A -85,B 0,C 180,E1 18388.112,E2 18388.112} C_VEL
LIN {X 0,Y 421.91,Z 512.912,A -85,B 0,C 180,E1 18385.627,E2 18385.627} C_VEL
LIN {X 0,Y 414.766,Z 503.349,A -85,B 0,C 180,E1 18382.838,E2 18382.838} C_VEL
LIN {X 0,Y 407.684,Z 494.073,A -85,B 0,C 180,E1 18379.559,E2 18379.559} C_VEL
LIN {X 0,Y 404.025,Z 489.604,A -85,B 0,C 180,E1 18377.574,E2 18377.574} C_VEL
LIN {X 0,Y 402.419,Z 487.582,A -85,B 0,C 180,E1 18376.603,E2 18376.603} C_VEL
LIN {X 0,Y 398.379,Z 482.633,A -85,B 0,C 180,E1 18373.795,E2 18373.795} C_VEL
LIN {X 0,Y 394.747,Z 477.313,A -85,B 0,C 180,E1 18369.918,E2 18369.918} C_VEL
LIN {X 0,Y 392.519,Z 473.83,A -85,B 0,C 180,E1 18363.798,E2 18363.798} C_VEL
LIN {X 0,Y 392.362,Z 473.126,A -85,B 0,C 180,E1 18360.146,E2 18360.146} C_VEL
LIN {X 0,Y 392.682,Z 474.139,A -85,B 0,C 180,E1 18356.496,E2 18356.496} C_VEL
LIN {X 0,Y 397.985,Z 479.236,A -85,B 0,C 180,E1 18350.455,E2 18350.455} C_VEL
LIN {X 0,Y 403.013,Z 484.67,A -85,B 0,C 180,E1 18346.952,E2 18346.952} C_VEL
LIN {X 0,Y 409.863,Z 492.398,A -85,B 0,C 180,E1 18343.269,E2 18343.269} C_VEL
LIN {X 0,Y 415.355,Z 498.929,A -85,B 0,C 180,E1 18340.816,E2 18340.816} C_VEL
LIN {X 0,Y 422.459,Z 507.431,A -85,B 0,C 180,E1 18338.076,E2 18338.076} C_VEL
LIN {X 0,Y 430.797,Z 518.211,A -85,B 0,C 180,E1 18335.269,E2 18335.269} C_VEL
LIN {X 0,Y 438.666,Z 528.966,A -85,B 0,C 180,E1 18332.915,E2 18332.915} C_VEL
LIN {X 0,Y 447.106,Z 540.997,A -85,B 0,C 180,E1 18330.638,E2 18330.638} C_VEL
LIN {X 0,Y 457.582,Z 557.13,A -85,B 0,C 180,E1 18328.075,E2 18328.075} C_VEL
LIN {X 0,Y 467.883,Z 574.48,A -85,B 0,C 180,E1 18325.77,E2 18325.77} C_VEL
LIN {X 0,Y 454.989,Z 798.129,A -85,B 0,C 180,E1 18322.097,E2 18322.097} C_VEL
LIN {X 0,Y 451.966,Z 847.51,A -85,B 0,C 180,E1 18321.248,E2 18321.248} C_VEL
LIN {X 0,Y 449.24,Z 871.555,A -85,B 0,C 180,E1 18320.658,E2 18320.658} C_VEL
LIN {X 0,Y 445.897,Z 894.445,A -85,B 0,C 180,E1 18319.926,E2 18319.926} C_VEL
LIN {X 0,Y 441.609,Z 917.565,A -85,B 0,C 180,E1 18318.957,E2 18318.957} C_VEL
LIN {X 0,Y 437.013,Z 939.234,A -85,B 0,C 180,E1 18317.844,E2 18317.844} C_VEL
LIN {X 0,Y 431.626,Z 960.962,A -85,B 0,C 180,E1 18316.476,E2 18316.476} C_VEL
LIN {X 0,Y 426.511,Z 979.828,A -85,B 0,C 180,E1 18315.072,E2 18315.072} C_VEL
LIN {X 0,Y 420.124,Z 1001.251,A -85,B 0,C 180,E1 18313.177,E2 18313.177} C_VEL
LIN {X 0,Y 414.377,Z 1019.288,A -85,B 0,C 180,E1 18311.297,E2 18311.297} C_VEL
LIN {X 0,Y 407.764,Z 1038.889,A -85,B 0,C 180,E1 18308.884,E2 18308.884} C_VEL
LIN {X 0,Y 402.256,Z 1054.782,A -85,B 0,C 180,E1 18306.593,E2 18306.593} C_VEL
LIN {X 0,Y 396.291,Z 1071.748,A -85,B 0,C 180,E1 18303.717,E2 18303.717} C_VEL
LIN {X 0,Y 391.591,Z 1085.219,A -85,B 0,C 180,E1 18301.05,E2 18301.05} C_VEL
LIN {X 0,Y 386.812,Z 1099.435,A -85,B 0,C 180,E1 18297.729,E2 18297.729} C_VEL
LIN {X 0,Y 383.325,Z 1110.548,A -85,B 0,C 180,E1 18294.668,E2 18294.668} C_VEL
LIN {X 0,Y 380.276,Z 1121.333,A -85,B 0,C 180,E1 18291.114,E2 18291.114} C_VEL
LIN {X 0,Y 378.368,Z 1129.315,A -85,B 0,C 180,E1 18287.945,E2 18287.945} C_VEL
LIN {X 0,Y 376.922,Z 1137.072,A -85,B 0,C 180,E1 18284.126,E2 18284.126} C_VEL
LIN {X 0,Y 376.262,Z 1142.147,A -85,B 0,C 180,E1 18280.876,E2 18280.876} C_VEL
LIN {X 0,Y 375.977,Z 1146.256,A -85,B 0,C 180,E1 18277.334,E2 18277.334} C_VEL
LIN {X 0,Y 375.953,Z 1148.561,A -85,B 0,C 180,E1 18273.965,E2 18273.965} C_VEL
LIN {X 0,Y 375.959,Z 1149.474,A -85,B 0,C 180,E1 18271.067,E2 18271.067} C_VEL
LIN {X 0,Y 375.958,Z 1149.329,A -85,B 0,C 180,E1 18268.019,E2 18268.019} C_VEL
LIN {X 0,Y 375.937,Z 1147.67,A -85,B 0,C 180,E1 18264.505,E2 18264.505} C_VEL
LIN {X 0,Y 376.049,Z 1144.939,A -85,B 0,C 180,E1 18261.437,E2 18261.437} C_VEL
LIN {X 0,Y 376.394,Z 1140.841,A -85,B 0,C 180,E1 18258.197,E2 18258.197} C_VEL
LIN {X 0,Y 377.346,Z 1134.428,A -85,B 0,C 180,E1 18254.477,E2 18254.477} C_VEL
LIN {X 0,Y 378.721,Z 1127.669,A -85,B 0,C 180,E1 18251.37,E2 18251.37} C_VEL
LIN {X 0,Y 381.105,Z 1118.254,A -85,B 0,C 180,E1 18247.802,E2 18247.802} C_VEL
LIN {X 0,Y 384.114,Z 1107.855,A -85,B 0,C 180,E1 18244.563,E2 18244.563} C_VEL
LIN {X 0,Y 388.217,Z 1095.133,A -85,B 0,C 180,E1 18241.207,E2 18241.207} C_VEL
LIN {X 0,Y 392.74,Z 1081.779,A -85,B 0,C 180,E1 18238.249,E2 18238.249} C_VEL
LIN {X 0,Y 398.28,Z 1065.969,A -85,B 0,C 180,E1 18235.257,E2 18235.257} C_VEL
LIN {X 0,Y 403.609,Z 1050.729,A -85,B 0,C 180,E1 18232.808,E2 18232.808} C_VEL
LIN {X 0,Y 409.834,Z 1032.762,A -85,B 0,C 180,E1 18230.326,E2 18230.326} C_VEL
LIN {X 0,Y 415.557,Z 1015.423,A -85,B 0,C 180,E1 18228.294,E2 18228.294} C_VEL
LIN {X 0,Y 421.808,Z 995.658,A -85,B 0,C 180,E1 18226.303,E2 18226.303} C_VEL
LIN {X 0,Y 427.611,Z 975.497,A -85,B 0,C 180,E1 18224.6,E2 18224.6} C_VEL
LIN {X 0,Y 433.294,Z 954.309,A -85,B 0,C 180,E1 18223.084,E2 18223.084} C_VEL
LIN {X 0,Y 438.463,Z 932.086,A -85,B 0,C 180,E1 18221.78,E2 18221.78} C_VEL
LIN {X 0,Y 443.095,Z 909.649,A -85,B 0,C 180,E1 18220.692,E2 18220.692} C_VEL
LIN {X 0,Y 446.992,Z 886.542,A -85,B 0,C 180,E1 18219.816,E2 18219.816} C_VEL
LIN {X 0,Y 450.242,Z 863.116,A -85,B 0,C 180,E1 18219.121,E2 18219.121} C_VEL
LIN {X 0,Y 452.496,Z 838.699,A -85,B 0,C 180,E1 18218.6,E2 18218.6} C_VEL
LIN {X 0,Y 465.802,Z 607.767,A -85,B 0,C 180,E1 18214.784,E2 18214.784} C_VEL
LIN {X 0,Y 467.656,Z 574.201,A -85,B 0,C 180,E1 18214.216,E2 18214.216} C_VEL
LIN {X 0,Y 456.974,Z 556.227,A -85,B 0,C 180,E1 18211.825,E2 18211.825} C_VEL
LIN {X 0,Y 445.74,Z 538.974,A -85,B 0,C 180,E1 18209.056,E2 18209.056} C_VEL
LIN {X 0,Y 436.632,Z 526.167,A -85,B 0,C 180,E1 18206.559,E2 18206.559} C_VEL
LIN {X 0,Y 428.873,Z 515.818,A -85,B 0,C 180,E1 18204.189,E2 18204.189} C_VEL
LIN {X 0,Y 423.939,Z 509.513,A -85,B 0,C 180,E1 18202.536,E2 18202.536} C_VEL
LIN {X 0,Y 417.401,Z 501.365,A -85,B 0,C 180,E1 18200.106,E2 18200.106} C_VEL
LIN {X 0,Y 412.672,Z 495.814,A -85,B 0,C 180,E1 18198.141,E2 18198.141} C_VEL
LIN {X 0,Y 408.118,Z 490.457,A -85,B 0,C 180,E1 18195.999,E2 18195.999} C_VEL
LIN {X 0,Y 402.995,Z 484.637,A -85,B 0,C 180,E1 18193.195,E2 18193.195} C_VEL
LIN {X 0,Y 397.723,Z 478.892,A -85,B 0,C 180,E1 18189.551,E2 18189.551} C_VEL
LIN {X 0,Y 392.642,Z 473.963,A -85,B 0,C 180,E1 18183.796,E2 18183.796} C_VEL
LIN {X 0,Y 392.238,Z 472.826,A -85,B 0,C 180,E1 18180.292,E2 18180.292} C_VEL
LIN {X 0,Y 392.32,Z 473.265,A -85,B 0,C 180,E1 18176.786,E2 18176.786} C_VEL
LIN {X 0,Y 393.601,Z 475.995,A -85,B 0,C 180,E1 18171.674,E2 18171.674} C_VEL
LIN {X 0,Y 394.948,Z 477.765,A -85,B 0,C 180,E1 18169.35,E2 18169.35} C_VEL
LIN {X 0,Y 398.375,Z 482.631,A -85,B 0,C 180,E1 18165.909,E2 18165.909} C_VEL
LIN {X 0,Y 403.655,Z 489.041,A -85,B 0,C 180,E1 18162.41,E2 18162.41} C_VEL
LIN {X 0,Y 407.146,Z 493.586,A -85,B 0,C 180,E1 18160.488,E2 18160.488} C_VEL
LIN {X 0,Y 412.667,Z 500.787,A -85,B 0,C 180,E1 18157.866,E2 18157.866} C_VEL
LIN {X 0,Y 416.355,Z 505.52,A -85,B 0,C 180,E1 18156.318,E2 18156.318} C_VEL
LIN {X 0,Y 423.362,Z 515.09,A -85,B 0,C 180,E1 18153.677,E2 18153.677} C_VEL
LIN {X 0,Y 428.282,Z 521.954,A -85,B 0,C 180,E1 18152.013,E2 18152.013} C_VEL
LIN {X 0,Y 433.592,Z 529.649,A -85,B 0,C 180,E1 18150.353,E2 18150.353} C_VEL
LIN {X 0,Y 440.479,Z 539.798,A -85,B 0,C 180,E1 18148.374,E2 18148.374} C_VEL
LIN {X 0,Y 451.229,Z 557.054,A -85,B 0,C 180,E1 18145.574,E2 18145.574} C_VEL
LIN {X 0,Y 461.507,Z 575.011,A -85,B 0,C 180,E1 18143.159,E2 18143.159} C_VEL
LIN {X 0,Y 465.875,Z 583.366,A -85,B 0,C 180,E1 18142.189,E2 18142.189} C_VEL
LIN {X 0,Y 452.786,Z 832.824,A -85,B 0,C 180,E1 18138.281,E2 18138.281} C_VEL
LIN {X 0,Y 450.901,Z 857.311,A -85,B 0,C 180,E1 18137.823,E2 18137.823} C_VEL
LIN {X 0,Y 448.104,Z 880.689,A -85,B 0,C 180,E1 18137.222,E2 18137.222} C_VEL
LIN {X 0,Y 444.578,Z 902.526,A -85,B 0,C 180,E1 18136.45,E2 18136.45} C_VEL
LIN {X 0,Y 440.354,Z 924.387,A -85,B 0,C 180,E1 18135.479,E2 18135.479} C_VEL
LIN {X 0,Y 435.38,Z 945.8,A -85,B 0,C 180,E1 18134.28,E2 18134.28} C_VEL
LIN {X 0,Y 429.655,Z 967.444,A -85,B 0,C 180,E1 18132.808,E2 18132.808} C_VEL
LIN {X 0,Y 424.21,Z 985.832,A -85,B 0,C 180,E1 18131.299,E2 18131.299} C_VEL
LIN {X 0,Y 417.615,Z 1006.278,A -85,B 0,C 180,E1 18129.293,E2 18129.293} C_VEL
LIN {X 0,Y 411.875,Z 1022.827,A -85,B 0,C 180,E1 18127.367,E2 18127.367} C_VEL
LIN {X 0,Y 405.686,Z 1039.679,A -85,B 0,C 180,E1 18125.049,E2 18125.049} C_VEL
LIN {X 0,Y 400.009,Z 1054.738,A -85,B 0,C 180,E1 18122.606,E2 18122.606} C_VEL
LIN {X 0,Y 394.398,Z 1069.287,A -85,B 0,C 180,E1 18119.796,E2 18119.796} C_VEL
LIN {X 0,Y 389.535,Z 1082.171,A -85,B 0,C 180,E1 18116.858,E2 18116.858} C_VEL
LIN {X 0,Y 385.324,Z 1093.516,A -85,B 0,C 180,E1 18113.717,E2 18113.717} C_VEL
LIN {X 0,Y 381.894,Z 1103.602,A -85,B 0,C 180,E1 18110.379,E2 18110.379} C_VEL
LIN {X 0,Y 379.476,Z 1111.436,A -85,B 0,C 180,E1 18107.164,E2 18107.164} C_VEL
LIN {X 0,Y 377.696,Z 1118.393,A -85,B 0,C 180,E1 18103.628,E2 18103.628} C_VEL
LIN {X 0,Y 376.691,Z 1123.372,A -85,B 0,C 180,E1 18100.244,E2 18100.244} C_VEL
LIN {X 0,Y 376.178,Z 1127.101,A -85,B 0,C 180,E1 18096.716,E2 18096.716} C_VEL
LIN {X 0,Y 376.004,Z 1129.064,A -85,B 0,C 180,E1 18093.507,E2 18093.507} C_VEL
LIN {X 0,Y 375.974,Z 1129.866,A -85,B 0,C 180,E1 18090.305,E2 18090.305} C_VEL
LIN {X 0,Y 375.997,Z 1129.24,A -85,B 0,C 180,E1 18086.799,E2 18086.799} C_VEL
LIN {X 0,Y 376.133,Z 1127.504,A -85,B 0,C 180,E1 18083.743,E2 18083.743} C_VEL
LIN {X 0,Y 376.603,Z 1123.907,A -85,B 0,C 180,E1 18080.062,E2 18080.062} C_VEL
LIN {X 0,Y 377.489,Z 1119.297,A -85,B 0,C 180,E1 18076.833,E2 18076.833} C_VEL
LIN {X 0,Y 379.238,Z 1112.354,A -85,B 0,C 180,E1 18073.141,E2 18073.141} C_VEL
LIN {X 0,Y 381.554,Z 1104.653,A -85,B 0,C 180,E1 18069.922,E2 18069.922} C_VEL
LIN {X 0,Y 385.056,Z 1094.347,A -85,B 0,C 180,E1 18066.428,E2 18066.428} C_VEL
LIN {X 0,Y 386.118,Z 1091.414,A -85,B 0,C 180,E1 18065.547,E2 18065.547} C_VEL
LIN {X 0,Y 386.472,Z 1088.059,A -85,B 0,C 180,E1 18064.51,E2 18064.51} C_VEL
LIN {X 0,Y 384.337,Z 1078.866,A -85,B 0,C 180,E1 18061.681,E2 18061.681} C_VEL
LIN {X 0,Y 385.006,Z 1075.555,A -85,B 0,C 180,E1 18060.825,E2 18060.825} C_VEL
LIN {X 0,Y 390.384,Z 1062.064,A -85,B 0,C 180,E1 18057.973,E2 18057.973} C_VEL
LIN {X 0,Y 396.232,Z 1047.477,A -85,B 0,C 180,E1 18055.352,E2 18055.352} C_VEL
LIN {X 0,Y 402.576,Z 1030.937,A -85,B 0,C 180,E1 18052.871,E2 18052.871} C_VEL
LIN {X 0,Y 408.908,Z 1013.955,A -85,B 0,C 180,E1 18050.704,E2 18050.704} C_VEL
LIN {X 0,Y 415.089,Z 995.975,A -85,B 0,C 180,E1 18048.79,E2 18048.79} C_VEL
LIN {X 0,Y 421.234,Z 976.873,A -85,B 0,C 180,E1 18047.058,E2 18047.058} C_VEL
LIN {X 0,Y 426.824,Z 957.443,A -85,B 0,C 180,E1 18045.603,E2 18045.603} C_VEL
LIN {X 0,Y 432.273,Z 936.409,A -85,B 0,C 180,E1 18044.282,E2 18044.282} C_VEL
LIN {X 0,Y 436.667,Z 916.454,A -85,B 0,C 180,E1 18043.267,E2 18043.267} C_VEL
LIN {X 0,Y 440.861,Z 894.397,A -85,B 0,C 180,E1 18042.353,E2 18042.353} C_VEL
LIN {X 0,Y 444.113,Z 872.206,A -85,B 0,C 180,E1 18041.658,E2 18041.658} C_VEL
LIN {X 0,Y 446.712,Z 848.759,A -85,B 0,C 180,E1 18041.11,E2 18041.11} C_VEL
LIN {X 0,Y 450.211,Z 786.57,A -85,B 0,C 180,E1 18040.101,E2 18040.101} C_VEL
LIN {X 0,Y 461.079,Z 586.757,A -85,B 0,C 180,E1 18036.942,E2 18036.942} C_VEL
LIN {X 0,Y 452.134,Z 570.42,A -85,B 0,C 180,E1 18034.848,E2 18034.848} C_VEL
LIN {X 0,Y 443.698,Z 556.138,A -85,B 0,C 180,E1 18032.703,E2 18032.703} C_VEL
LIN {X 0,Y 434.663,Z 541.802,A -85,B 0,C 180,E1 18030.175,E2 18030.175} C_VEL
LIN {X 0,Y 426.677,Z 529.977,A -85,B 0,C 180,E1 18027.684,E2 18027.684} C_VEL
LIN {X 0,Y 419.381,Z 519.595,A -85,B 0,C 180,E1 18025.112,E2 18025.112} C_VEL
LIN {X 0,Y 412.873,Z 510.732,A -85,B 0,C 180,E1 18022.498,E2 18022.498} C_VEL
LIN {X 0,Y 405.924,Z 501.522,A -85,B 0,C 180,E1 18019.199,E2 18019.199} C_VEL
LIN {X 0,Y 402.363,Z 496.977,A -85,B 0,C 180,E1 18017.201,E2 18017.201} C_VEL
LIN {X 0,Y 397.234,Z 490.519,A -85,B 0,C 180,E1 18013.683,E2 18013.683} C_VEL
LIN {X 0,Y 393.105,Z 485.043,A -85,B 0,C 180,E1 18009.664,E2 18009.664} C_VEL
LIN {X 0,Y 390.065,Z 481.376,A -85,B 0,C 180,E1 18003.527,E2 18003.527} C_VEL
LIN {X 0,Y 390.157,Z 480.844,A -85,B 0,C 180,E1 18000,E2 18000} C_VEL
LIN {X 0,Y 391.597,Z 482.159,A -85,B 0,C 180,E1 17996.34,E2 17996.34} C_VEL
LIN {X 0,Y 396.824,Z 487.144,A -85,B 0,C 180,E1 17990.573,E2 17990.573} C_VEL
LIN {X 0,Y 401.807,Z 492.551,A -85,B 0,C 180,E1 17987.058,E2 17987.058} C_VEL
LIN {X 0,Y 408.178,Z 499.938,A -85,B 0,C 180,E1 17983.565,E2 17983.565} C_VEL
LIN {X 0,Y 413.577,Z 506.482,A -85,B 0,C 180,E1 17981.097,E2 17981.097} C_VEL
LIN {X 0,Y 420.407,Z 514.813,A -85,B 0,C 180,E1 17978.404,E2 17978.404} C_VEL
LIN {X 0,Y 428.434,Z 525.352,A -85,B 0,C 180,E1 17975.638,E2 17975.638} C_VEL
LIN {X 0,Y 436.289,Z 536.274,A -85,B 0,C 180,E1 17973.234,E2 17973.234} C_VEL
LIN {X 0,Y 444.406,Z 548.044,A -85,B 0,C 180,E1 17970.996,E2 17970.996} C_VEL
LIN {X 0,Y 454.625,Z 564.089,A -85,B 0,C 180,E1 17968.436,E2 17968.436} C_VEL
LIN {X 0,Y 462.976,Z 578.452,A -85,B 0,C 180,E1 17966.507,E2 17966.507} C_VEL
LIN {X 0,Y 449.54,Z 804.732,A -85,B 0,C 180,E1 17962.774,E2 17962.774} C_VEL
LIN {X 0,Y 446.766,Z 848.01,A -85,B 0,C 180,E1 17962.02,E2 17962.02} C_VEL
LIN {X 0,Y 443.99,Z 871.824,A -85,B 0,C 180,E1 17961.433,E2 17961.433} C_VEL
LIN {X 0,Y 440.586,Z 894.513,A -85,B 0,C 180,E1 17960.704,E2 17960.704} C_VEL
LIN {X 0,Y 436.257,Z 917.264,A -85,B 0,C 180,E1 17959.75,E2 17959.75} C_VEL
LIN {X 0,Y 431.578,Z 938.724,A -85,B 0,C 180,E1 17958.647,E2 17958.647} C_VEL
LIN {X 0,Y 426.037,Z 960.545,A -85,B 0,C 180,E1 17957.274,E2 17957.274} C_VEL
LIN {X 0,Y 420.754,Z 979.443,A -85,B 0,C 180,E1 17955.864,E2 17955.864} C_VEL
LIN {X 0,Y 414.169,Z 1000.917,A -85,B 0,C 180,E1 17953.955,E2 17953.955} C_VEL
LIN {X 0,Y 408.347,Z 1018.585,A -85,B 0,C 180,E1 17952.103,E2 17952.103} C_VEL
LIN {X 0,Y 401.546,Z 1038.086,A -85,B 0,C 180,E1 17949.696,E2 17949.696} C_VEL
LIN {X 0,Y 395.901,Z 1053.736,A -85,B 0,C 180,E1 17947.427,E2 17947.427} C_VEL
LIN {X 0,Y 389.707,Z 1070.702,A -85,B 0,C 180,E1 17944.544,E2 17944.544} C_VEL
LIN {X 0,Y 384.754,Z 1084.249,A -85,B 0,C 180,E1 17941.84,E2 17941.84} C_VEL
LIN {X 0,Y 379.565,Z 1098.96,A -85,B 0,C 180,E1 17938.374,E2 17938.374} C_VEL
LIN {X 0,Y 375.97,Z 1109.782,A -85,B 0,C 180,E1 17935.352,E2 17935.352} C_VEL
LIN {X 0,Y 372.583,Z 1121.106,A -85,B 0,C 180,E1 17931.572,E2 17931.572} C_VEL
LIN {X 0,Y 370.586,Z 1128.94,A -85,B 0,C 180,E1 17928.402,E2 17928.402} C_VEL
LIN {X 0,Y 369.046,Z 1136.59,A -85,B 0,C 180,E1 17924.594,E2 17924.594} C_VEL
LIN {X 0,Y 368.317,Z 1141.717,A -85,B 0,C 180,E1 17921.272,E2 17921.272} C_VEL
LIN {X 0,Y 367.995,Z 1145.571,A -85,B 0,C 180,E1 17917.965,E2 17917.965} C_VEL
LIN {X 0,Y 367.952,Z 1148.208,A -85,B 0,C 180,E1 17914.364,E2 17914.364} C_VEL
LIN {X 0,Y 367.963,Z 1149.24,A -85,B 0,C 180,E1 17911.246,E2 17911.246} C_VEL
LIN {X 0,Y 367.962,Z 1149.167,A -85,B 0,C 180,E1 17908.287,E2 17908.287} C_VEL
LIN {X 0,Y 367.935,Z 1147.694,A -85,B 0,C 180,E1 17904.698,E2 17904.698} C_VEL
LIN {X 0,Y 368.05,Z 1144.891,A -85,B 0,C 180,E1 17901.407,E2 17901.407} C_VEL
LIN {X 0,Y 368.384,Z 1141.054,A -85,B 0,C 180,E1 17898.254,E2 17898.254} C_VEL
LIN {X 0,Y 369.348,Z 1134.833,A -85,B 0,C 180,E1 17894.454,E2 17894.454} C_VEL
LIN {X 0,Y 370.842,Z 1127.808,A -85,B 0,C 180,E1 17891.122,E2 17891.122} C_VEL
LIN {X 0,Y 373.289,Z 1118.658,A -85,B 0,C 180,E1 17887.536,E2 17887.536} C_VEL
LIN {X 0,Y 376.474,Z 1108.146,A -85,B 0,C 180,E1 17884.178,E2 17884.178} C_VEL
LIN {X 0,Y 380.53,Z 1096.181,A -85,B 0,C 180,E1 17880.915,E2 17880.915} C_VEL
LIN {X 0,Y 385.26,Z 1082.735,A -85,B 0,C 180,E1 17877.856,E2 17877.856} C_VEL
LIN {X 0,Y 390.606,Z 1068.196,A -85,B 0,C 180,E1 17875,E2 17875} C_VEL
LIN {X 0,Y 396.523,Z 1051.862,A -85,B 0,C 180,E1 17872.302,E2 17872.302} C_VEL
LIN {X 0,Y 402.872,Z 1034.334,A -85,B 0,C 180,E1 17869.812,E2 17869.812} C_VEL
LIN {X 0,Y 409.23,Z 1015.716,A -85,B 0,C 180,E1 17867.595,E2 17867.595} C_VEL
LIN {X 0,Y 415.627,Z 996.213,A -85,B 0,C 180,E1 17865.603,E2 17865.603} C_VEL
LIN {X 0,Y 421.655,Z 975.924,A -85,B 0,C 180,E1 17863.872,E2 17863.872} C_VEL
LIN {X 0,Y 427.515,Z 954.798,A -85,B 0,C 180,E1 17862.345,E2 17862.345} C_VEL
LIN {X 0,Y 432.816,Z 932.702,A -85,B 0,C 180,E1 17861.037,E2 17861.037} C_VEL
LIN {X 0,Y 437.541,Z 910.576,A -85,B 0,C 180,E1 17859.953,E2 17859.953} C_VEL
LIN {X 0,Y 441.635,Z 887.055,A -85,B 0,C 180,E1 17859.052,E2 17859.052} C_VEL
LIN {X 0,Y 444.933,Z 864.034,A -85,B 0,C 180,E1 17858.363,E2 17858.363} C_VEL
LIN {X 0,Y 447.302,Z 839.461,A -85,B 0,C 180,E1 17857.831,E2 17857.831} C_VEL
LIN {X 0,Y 460.929,Z 610.02,A -85,B 0,C 180,E1 17854.021,E2 17854.021} C_VEL
LIN {X 0,Y 462.733,Z 578.039,A -85,B 0,C 180,E1 17853.474,E2 17853.474} C_VEL
LIN {X 0,Y 453.321,Z 562.055,A -85,B 0,C 180,E1 17851.295,E2 17851.295} C_VEL
LIN {X 0,Y 442.401,Z 545.031,A -85,B 0,C 180,E1 17848.519,E2 17848.519} C_VEL
LIN {X 0,Y 433.363,Z 532.214,A -85,B 0,C 180,E1 17845.964,E2 17845.964} C_VEL
LIN {X 0,Y 426.155,Z 522.47,A -85,B 0,C 180,E1 17843.691,E2 17843.691} C_VEL
LIN {X 0,Y 419.949,Z 514.268,A -85,B 0,C 180,E1 17841.511,E2 17841.511} C_VEL
LIN {X 0,Y 411.852,Z 504.222,A -85,B 0,C 180,E1 17838.251,E2 17838.251} C_VEL
LIN {X 0,Y 406.456,Z 498.016,A -85,B 0,C 180,E1 17835.7,E2 17835.7} C_VEL
LIN {X 0,Y 401.55,Z 492.344,A -85,B 0,C 180,E1 17832.95,E2 17832.95} C_VEL
LIN {X 0,Y 396.042,Z 486.317,A -85,B 0,C 180,E1 17829.006,E2 17829.006} C_VEL
LIN {X 0,Y 390.974,Z 481.49,A -85,B 0,C 180,E1 17823.079,E2 17823.079} C_VEL
LIN {X 0,Y 389.743,Z 480.385,A -85,B 0,C 180,E1 17819.412,E2 17819.412} C_VEL
LIN {X 0,Y 389.846,Z 481.162,A -85,B 0,C 180,E1 17815.882,E2 17815.882} C_VEL
LIN {X 0,Y 393.359,Z 485.416,A -85,B 0,C 180,E1 17809.602,E2 17809.602} C_VEL
LIN {X 0,Y 398.066,Z 491.65,A -85,B 0,C 180,E1 17805.378,E2 17805.378} C_VEL
LIN {X 0,Y 402.214,Z 496.812,A -85,B 0,C 180,E1 17802.643,E2 17802.643} C_VEL
LIN {X 0,Y 405.796,Z 501.412,A -85,B 0,C 180,E1 17800.645,E2 17800.645} C_VEL
LIN {X 0,Y 411.177,Z 508.68,A -85,B 0,C 180,E1 17798.044,E2 17798.044} C_VEL
LIN {X 0,Y 414.425,Z 512.921,A -85,B 0,C 180,E1 17796.653,E2 17796.653} C_VEL
LIN {X 0,Y 421.146,Z 522.253,A -85,B 0,C 180,E1 17794.059,E2 17794.059} C_VEL
LIN {X 0,Y 427.321,Z 530.956,A -85,B 0,C 180,E1 17791.945,E2 17791.945} C_VEL
LIN {X 0,Y 435.477,Z 543.217,A -85,B 0,C 180,E1 17789.433,E2 17789.433} C_VEL
LIN {X 0,Y 444.508,Z 557.565,A -85,B 0,C 180,E1 17786.942,E2 17786.942} C_VEL
LIN {X 0,Y 453.949,Z 573.768,A -85,B 0,C 180,E1 17784.579,E2 17784.579} C_VEL
LIN {X 0,Y 461.008,Z 586.922,A -85,B 0,C 180,E1 17782.941,E2 17782.941} C_VEL
LIN {X 0,Y 447.532,Z 835.338,A -85,B 0,C 180,E1 17779.025,E2 17779.025} C_VEL
LIN {X 0,Y 445.583,Z 858.742,A -85,B 0,C 180,E1 17778.575,E2 17778.575} C_VEL
LIN {X 0,Y 442.527,Z 882.78,A -85,B 0,C 180,E1 17777.936,E2 17777.936} C_VEL
LIN {X 0,Y 438.99,Z 903.934,A -85,B 0,C 180,E1 17777.174,E2 17777.174} C_VEL
LIN {X 0,Y 434.262,Z 927.151,A -85,B 0,C 180,E1 17776.111,E2 17776.111} C_VEL
LIN {X 0,Y 429.431,Z 947.261,A -85,B 0,C 180,E1 17774.965,E2 17774.965} C_VEL
LIN {X 0,Y 423.552,Z 968.633,A -85,B 0,C 180,E1 17773.484,E2 17773.484} C_VEL
LIN {X 0,Y 417.964,Z 986.917,A -85,B 0,C 180,E1 17771.963,E2 17771.963} C_VEL
LIN {X 0,Y 411.389,Z 1006.592,A -85,B 0,C 180,E1 17770.007,E2 17770.007} C_VEL
LIN {X 0,Y 405.464,Z 1023.126,A -85,B 0,C 180,E1 17768.062,E2 17768.062} C_VEL
LIN {X 0,Y 399.064,Z 1039.953,A -85,B 0,C 180,E1 17765.719,E2 17765.719} C_VEL
LIN {X 0,Y 393.306,Z 1054.649,A -85,B 0,C 180,E1 17763.308,E2 17763.308} C_VEL
LIN {X 0,Y 387.491,Z 1069.172,A -85,B 0,C 180,E1 17760.473,E2 17760.473} C_VEL
LIN {X 0,Y 382.501,Z 1081.795,A -85,B 0,C 180,E1 17757.561,E2 17757.561} C_VEL
LIN {X 0,Y 378.051,Z 1093.247,A -85,B 0,C 180,E1 17754.368,E2 17754.368} C_VEL
LIN {X 0,Y 374.407,Z 1103.434,A -85,B 0,C 180,E1 17750.969,E2 17750.969} C_VEL
LIN {X 0,Y 371.709,Z 1111.658,A -85,B 0,C 180,E1 17747.534,E2 17747.534} C_VEL
LIN {X 0,Y 369.815,Z 1118.624,A -85,B 0,C 180,E1 17743.915,E2 17743.915} C_VEL
LIN {X 0,Y 368.751,Z 1123.587,A -85,B 0,C 180,E1 17740.467,E2 17740.467} C_VEL
LIN {X 0,Y 368.196,Z 1127.313,A -85,B 0,C 180,E1 17736.863,E2 17736.863} C_VEL
LIN {X 0,Y 368.009,Z 1129.274,A -85,B 0,C 180,E1 17733.583,E2 17733.583} C_VEL
LIN {X 0,Y 367.977,Z 1130.075,A -85,B 0,C 180,E1 17730.311,E2 17730.311} C_VEL
LIN {X 0,Y 368.002,Z 1129.45,A -85,B 0,C 180,E1 17726.729,E2 17726.729} C_VEL
LIN {X 0,Y 368.149,Z 1127.714,A -85,B 0,C 180,E1 17723.607,E2 17723.607} C_VEL
LIN {X 0,Y 368.656,Z 1124.121,A -85,B 0,C 180,E1 17719.846,E2 17719.846} C_VEL
LIN {X 0,Y 369.6,Z 1119.512,A -85,B 0,C 180,E1 17716.546,E2 17716.546} C_VEL
LIN {X 0,Y 371.46,Z 1112.575,A -85,B 0,C 180,E1 17712.777,E2 17712.777} C_VEL
LIN {X 0,Y 373.906,Z 1104.875,A -85,B 0,C 180,E1 17709.493,E2 17709.493} C_VEL
LIN {X 0,Y 377.585,Z 1094.577,A -85,B 0,C 180,E1 17705.932,E2 17705.932} C_VEL
LIN {X 0,Y 381.69,Z 1083.911,A -85,B 0,C 180,E1 17702.882,E2 17702.882} C_VEL
LIN {X 0,Y 385.006,Z 1075.555,A -85,B 0,C 180,E1 17700.825,E2 17700.825} C_VEL
LIN {X 0,Y 385.751,Z 1071.612,A -85,B 0,C 180,E1 17699.836,E2 17699.836} C_VEL
LIN {X 0,Y 384.73,Z 1060.887,A -85,B 0,C 180,E1 17697.113,E2 17697.113} C_VEL
LIN {X 0,Y 385.712,Z 1057.095,A -85,B 0,C 180,E1 17696.313,E2 17696.313} C_VEL
LIN {X 0,Y 391.96,Z 1041.713,A -85,B 0,C 180,E1 17693.713,E2 17693.713} C_VEL
LIN {X 0,Y 398.539,Z 1025.208,A -85,B 0,C 180,E1 17691.339,E2 17691.339} C_VEL
LIN {X 0,Y 405.042,Z 1007.664,A -85,B 0,C 180,E1 17689.236,E2 17689.236} C_VEL
LIN {X 0,Y 411.743,Z 988.412,A -85,B 0,C 180,E1 17687.283,E2 17687.283} C_VEL
LIN {X 0,Y 417.796,Z 969.216,A -85,B 0,C 180,E1 17685.667,E2 17685.667} C_VEL
LIN {X 0,Y 424.102,Z 946.953,A -85,B 0,C 180,E1 17684.118,E2 17684.118} C_VEL
LIN {X 0,Y 429.073,Z 926.794,A -85,B 0,C 180,E1 17682.968,E2 17682.968} C_VEL
LIN {X 0,Y 433.8,Z 904.2,A -85,B 0,C 180,E1 17681.933,E2 17681.933} C_VEL
LIN {X 0,Y 437.475,Z 882.816,A -85,B 0,C 180,E1 17681.162,E2 17681.162} C_VEL
LIN {X 0,Y 440.613,Z 858.8,A -85,B 0,C 180,E1 17680.522,E2 17680.522} C_VEL
LIN {X 0,Y 442.604,Z 835.594,A -85,B 0,C 180,E1 17680.073,E2 17680.073} C_VEL
LIN {X 0,Y 456.356,Z 590.568,A -85,B 0,C 180,E1 17676.193,E2 17676.193} C_VEL
LIN {X 0,Y 447.205,Z 573.855,A -85,B 0,C 180,E1 17673.963,E2 17673.963} C_VEL
LIN {X 0,Y 438.585,Z 559.144,A -85,B 0,C 180,E1 17671.664,E2 17671.664} C_VEL
LIN {X 0,Y 430.256,Z 545.915,A -85,B 0,C 180,E1 17669.211,E2 17669.211} C_VEL
LIN {X 0,Y 423.098,Z 535.288,A -85,B 0,C 180,E1 17666.871,E2 17666.871} C_VEL
LIN {X 0,Y 415.23,Z 523.938,A -85,B 0,C 180,E1 17663.939,E2 17663.939} C_VEL
LIN {X 0,Y 410.536,Z 517.579,A -85,B 0,C 180,E1 17661.954,E2 17661.954} C_VEL
LIN {X 0,Y 404.445,Z 509.219,A -85,B 0,C 180,E1 17658.972,E2 17658.972} C_VEL
LIN {X 0,Y 400.826,Z 504.543,A -85,B 0,C 180,E1 17656.895,E2 17656.895} C_VEL
LIN {X 0,Y 395.917,Z 498.248,A -85,B 0,C 180,E1 17653.435,E2 17653.435} C_VEL
LIN {X 0,Y 391.899,Z 492.832,A -85,B 0,C 180,E1 17649.398,E2 17649.398} C_VEL
LIN {X 0,Y 389.073,Z 489.279,A -85,B 0,C 180,E1 17643.389,E2 17643.389} C_VEL
LIN {X 0,Y 389.207,Z 488.819,A -85,B 0,C 180,E1 17639.853,E2 17639.853} C_VEL
LIN {X 0,Y 390.614,Z 490.143,A -85,B 0,C 180,E1 17636.331,E2 17636.331} C_VEL
LIN {X 0,Y 395.582,Z 494.94,A -85,B 0,C 180,E1 17630.764,E2 17630.764} C_VEL
LIN {X 0,Y 401.264,Z 501.348,A -85,B 0,C 180,E1 17626.747,E2 17626.747} C_VEL
LIN {X 0,Y 406.635,Z 507.672,A -85,B 0,C 180,E1 17623.794,E2 17623.794} C_VEL
LIN {X 0,Y 411.809,Z 514.032,A -85,B 0,C 180,E1 17621.38,E2 17621.38} C_VEL
LIN {X 0,Y 418.37,Z 522.19,A -85,B 0,C 180,E1 17618.735,E2 17618.735} C_VEL
LIN {X 0,Y 425.996,Z 532.352,A -85,B 0,C 180,E1 17616.042,E2 17616.042} C_VEL
LIN {X 0,Y 434.132,Z 543.863,A -85,B 0,C 180,E1 17613.497,E2 17613.497} C_VEL
LIN {X 0,Y 442.052,Z 555.575,A -85,B 0,C 180,E1 17611.271,E2 17611.271} C_VEL
LIN {X 0,Y 452.383,Z 572.182,A -85,B 0,C 180,E1 17608.633,E2 17608.633} C_VEL
LIN {X 0,Y 458.138,Z 582.466,A -85,B 0,C 180,E1 17607.26,E2 17607.26} C_VEL
LIN {X 0,Y 444.326,Z 808.583,A -85,B 0,C 180,E1 17603.515,E2 17603.515} C_VEL
LIN {X 0,Y 441.65,Z 848.483,A -85,B 0,C 180,E1 17602.811,E2 17602.811} C_VEL
LIN {X 0,Y 438.84,Z 871.979,A -85,B 0,C 180,E1 17602.229,E2 17602.229} C_VEL
LIN {X 0,Y 435.418,Z 894.237,A -85,B 0,C 180,E1 17601.514,E2 17601.514} C_VEL
LIN {X 0,Y 431.049,Z 916.694,A -85,B 0,C 180,E1 17600.575,E2 17600.575} C_VEL
LIN {X 0,Y 426.465,Z 937.191,A -85,B 0,C 180,E1 17599.527,E2 17599.527} C_VEL
LIN {X 0,Y 420.534,Z 960.127,A -85,B 0,C 180,E1 17598.092,E2 17598.092} C_VEL
LIN {X 0,Y 415.082,Z 979.058,A -85,B 0,C 180,E1 17596.677,E2 17596.677} C_VEL
LIN {X 0,Y 408.252,Z 1000.706,A -85,B 0,C 180,E1 17594.743,E2 17594.743} C_VEL
LIN {X 0,Y 402.347,Z 1018.038,A -85,B 0,C 180,E1 17592.917,E2 17592.917} C_VEL
LIN {X 0,Y 395.026,Z 1038.315,A -85,B 0,C 180,E1 17590.39,E2 17590.39} C_VEL
LIN {X 0,Y 389.132,Z 1054.06,A -85,B 0,C 180,E1 17588.075,E2 17588.075} C_VEL
LIN {X 0,Y 382.589,Z 1071.231,A -85,B 0,C 180,E1 17585.097,E2 17585.097} C_VEL
LIN {X 0,Y 377.384,Z 1084.921,A -85,B 0,C 180,E1 17582.306,E2 17582.306} C_VEL
LIN {X 0,Y 372.193,Z 1098.955,A -85,B 0,C 180,E1 17578.919,E2 17578.919} C_VEL
LIN {X 0,Y 368.325,Z 1110.076,A -85,B 0,C 180,E1 17575.744,E2 17575.744} C_VEL
LIN {X 0,Y 364.915,Z 1120.879,A -85,B 0,C 180,E1 17572.048,E2 17572.048} C_VEL
LIN {X 0,Y 362.79,Z 1128.716,A -85,B 0,C 180,E1 17568.812,E2 17568.812} C_VEL
LIN {X 0,Y 361.135,Z 1136.378,A -85,B 0,C 180,E1 17564.918,E2 17564.918} C_VEL
LIN {X 0,Y 360.352,Z 1141.501,A -85,B 0,C 180,E1 17561.524,E2 17561.524} C_VEL
LIN {X 0,Y 360.007,Z 1145.358,A -85,B 0,C 180,E1 17558.143,E2 17558.143} C_VEL
LIN {X 0,Y 359.951,Z 1147.998,A -85,B 0,C 180,E1 17554.461,E2 17554.461} C_VEL
LIN {X 0,Y 359.966,Z 1149.031,A -85,B 0,C 180,E1 17551.273,E2 17551.273} C_VEL
LIN {X 0,Y 359.964,Z 1148.957,A -85,B 0,C 180,E1 17548.249,E2 17548.249} C_VEL
LIN {X 0,Y 359.937,Z 1147.482,A -85,B 0,C 180,E1 17544.58,E2 17544.58} C_VEL
LIN {X 0,Y 360.058,Z 1144.677,A -85,B 0,C 180,E1 17541.214,E2 17541.214} C_VEL
LIN {X 0,Y 360.424,Z 1140.837,A -85,B 0,C 180,E1 17537.991,E2 17537.991} C_VEL
LIN {X 0,Y 361.469,Z 1134.611,A -85,B 0,C 180,E1 17534.106,E2 17534.106} C_VEL
LIN {X 0,Y 363.063,Z 1127.583,A -85,B 0,C 180,E1 17530.702,E2 17530.702} C_VEL
LIN {X 0,Y 365.572,Z 1118.729,A -85,B 0,C 180,E1 17527.145,E2 17527.145} C_VEL
LIN {X 0,Y 369.026,Z 1107.908,A -85,B 0,C 180,E1 17523.617,E2 17523.617} C_VEL
LIN {X 0,Y 373.292,Z 1095.933,A -85,B 0,C 180,E1 17520.295,E2 17520.295} C_VEL
LIN {X 0,Y 378.254,Z 1082.48,A -85,B 0,C 180,E1 17517.186,E2 17517.186} C_VEL
LIN {X 0,Y 383.812,Z 1067.984,A -85,B 0,C 180,E1 17514.299,E2 17514.299} C_VEL
LIN {X 0,Y 390.085,Z 1051.37,A -85,B 0,C 180,E1 17511.525,E2 17511.525} C_VEL
LIN {X 0,Y 396.595,Z 1034.032,A -85,B 0,C 180,E1 17509.042,E2 17509.042} C_VEL
LIN {X 0,Y 403.18,Z 1015.393,A -85,B 0,C 180,E1 17506.805,E2 17506.805} C_VEL
LIN {X 0,Y 409.647,Z 996.309,A -85,B 0,C 180,E1 17504.841,E2 17504.841} C_VEL
LIN {X 0,Y 416.011,Z 975.529,A -85,B 0,C 180,E1 17503.057,E2 17503.057} C_VEL
LIN {X 0,Y 422.045,Z 954.362,A -85,B 0,C 180,E1 17501.526,E2 17501.526} C_VEL
LIN {X 0,Y 427.403,Z 932.629,A -85,B 0,C 180,E1 17500.237,E2 17500.237} C_VEL
LIN {X 0,Y 432.365,Z 909.933,A -85,B 0,C 180,E1 17499.125,E2 17499.125} C_VEL
LIN {X 0,Y 436.531,Z 886.491,A -85,B 0,C 180,E1 17498.232,E2 17498.232} C_VEL
LIN {X 0,Y 439.964,Z 862.855,A -85,B 0,C 180,E1 17497.531,E2 17497.531} C_VEL
LIN {X 0,Y 442.311,Z 838.645,A -85,B 0,C 180,E1 17497.014,E2 17497.014} C_VEL
LIN {X 0,Y 456.386,Z 608.3,A -85,B 0,C 180,E1 17493.176,E2 17493.176} C_VEL
LIN {X 0,Y 457.914,Z 581.921,A -85,B 0,C 180,E1 17492.721,E2 17492.721} C_VEL
LIN {X 0,Y 449.25,Z 567.14,A -85,B 0,C 180,E1 17490.643,E2 17490.643} C_VEL
LIN {X 0,Y 438.993,Z 550.951,A -85,B 0,C 180,E1 17487.946,E2 17487.946} C_VEL
LIN {X 0,Y 428.787,Z 536.199,A -85,B 0,C 180,E1 17484.929,E2 17484.929} C_VEL
LIN {X 0,Y 420.505,Z 525.105,A -85,B 0,C 180,E1 17482.141,E2 17482.141} C_VEL
LIN {X 0,Y 413.628,Z 516.253,A -85,B 0,C 180,E1 17479.487,E2 17479.487} C_VEL
LIN {X 0,Y 408.911,Z 510.572,A -85,B 0,C 180,E1 17477.43,E2 17477.43} C_VEL
LIN {X 0,Y 404.939,Z 505.696,A -85,B 0,C 180,E1 17475.467,E2 17475.467} C_VEL
LIN {X 0,Y 400.113,Z 500.049,A -85,B 0,C 180,E1 17472.704,E2 17472.704} C_VEL
LIN {X 0,Y 394.721,Z 494.072,A -85,B 0,C 180,E1 17468.742,E2 17468.742} C_VEL
LIN {X 0,Y 389.917,Z 489.376,A -85,B 0,C 180,E1 17462.94,E2 17462.94} C_VEL
LIN {X 0,Y 388.765,Z 488.325,A -85,B 0,C 180,E1 17459.411,E2 17459.411} C_VEL
LIN {X 0,Y 388.87,Z 489.133,A -85,B 0,C 180,E1 17455.871,E2 17455.871} C_VEL
LIN {X 0,Y 392.272,Z 493.349,A -85,B 0,C 180,E1 17449.708,E2 17449.708} C_VEL
LIN {X 0,Y 396.811,Z 499.497,A -85,B 0,C 180,E1 17445.554,E2 17445.554} C_VEL
LIN {X 0,Y 400.673,Z 504.378,A -85,B 0,C 180,E1 17442.949,E2 17442.949} C_VEL
LIN {X 0,Y 406.021,Z 511.507,A -85,B 0,C 180,E1 17439.982,E2 17439.982} C_VEL
LIN {X 0,Y 412.358,Z 520.076,A -85,B 0,C 180,E1 17437.059,E2 17437.059} C_VEL
LIN {X 0,Y 418.945,Z 529.409,A -85,B 0,C 180,E1 17434.445,E2 17434.445} C_VEL
LIN {X 0,Y 425.301,Z 538.552,A -85,B 0,C 180,E1 17432.219,E2 17432.219} C_VEL
LIN {X 0,Y 433.162,Z 550.619,A -85,B 0,C 180,E1 17429.748,E2 17429.748} C_VEL
LIN {X 0,Y 441.629,Z 564.367,A -85,B 0,C 180,E1 17427.356,E2 17427.356} C_VEL
LIN {X 0,Y 450.649,Z 580.116,A -85,B 0,C 180,E1 17425.04,E2 17425.04} C_VEL
LIN {X 0,Y 456.208,Z 590.641,A -85,B 0,C 180,E1 17423.705,E2 17423.705} C_VEL
LIN {X 0,Y 442.294,Z 838.149,A -85,B 0,C 180,E1 17419.778,E2 17419.778} C_VEL
LIN {X 0,Y 440.324,Z 860.366,A -85,B 0,C 180,E1 17419.341,E2 17419.341} C_VEL
LIN {X 0,Y 436.98,Z 885.131,A -85,B 0,C 180,E1 17418.658,E2 17418.658} C_VEL
LIN {X 0,Y 433.216,Z 906.761,A -85,B 0,C 180,E1 17417.86,E2 17417.86} C_VEL
LIN {X 0,Y 428.492,Z 928.786,A -85,B 0,C 180,E1 17416.822,E2 17416.822} C_VEL
LIN {X 0,Y 423.547,Z 948.718,A -85,B 0,C 180,E1 17415.669,E2 17415.669} C_VEL
LIN {X 0,Y 417.51,Z 969.822,A -85,B 0,C 180,E1 17414.18,E2 17414.18} C_VEL
LIN {X 0,Y 411.637,Z 988.442,A -85,B 0,C 180,E1 17412.608,E2 17412.608} C_VEL
LIN {X 0,Y 405.011,Z 1007.507,A -85,B 0,C 180,E1 17410.675,E2 17410.675} C_VEL
LIN {X 0,Y 398.515,Z 1025.066,A -85,B 0,C 180,E1 17408.572,E2 17408.572} C_VEL
LIN {X 0,Y 392.126,Z 1041.134,A -85,B 0,C 180,E1 17406.27,E2 17406.27} C_VEL
LIN {X 0,Y 385.877,Z 1056.567,A -85,B 0,C 180,E1 17403.678,E2 17403.678} C_VEL
LIN {X 0,Y 380.044,Z 1070.47,A -85,B 0,C 180,E1 17400.867,E2 17400.867} C_VEL
LIN {X 0,Y 374.799,Z 1083.224,A -85,B 0,C 180,E1 17397.831,E2 17397.831} C_VEL
LIN {X 0,Y 370.238,Z 1094.483,A -85,B 0,C 180,E1 17394.576,E2 17394.576} C_VEL
LIN {X 0,Y 366.351,Z 1104.837,A -85,B 0,C 180,E1 17390.949,E2 17390.949} C_VEL
LIN {X 0,Y 363.745,Z 1112.565,A -85,B 0,C 180,E1 17387.6,E2 17387.6} C_VEL
LIN {X 0,Y 361.753,Z 1119.563,A -85,B 0,C 180,E1 17383.751,E2 17383.751} C_VEL
LIN {X 0,Y 360.736,Z 1124.2,A -85,B 0,C 180,E1 17380.38,E2 17380.38} C_VEL
LIN {X 0,Y 360.171,Z 1127.851,A -85,B 0,C 180,E1 17376.536,E2 17376.536} C_VEL
LIN {X 0,Y 360.007,Z 1129.615,A -85,B 0,C 180,E1 17373.344,E2 17373.344} C_VEL
LIN {X 0,Y 359.978,Z 1130.3,A -85,B 0,C 180,E1 17369.682,E2 17369.682} C_VEL
LIN {X 0,Y 360.014,Z 1129.53,A -85,B 0,C 180,E1 17366.337,E2 17366.337} C_VEL
LIN {X 0,Y 360.208,Z 1127.599,A -85,B 0,C 180,E1 17362.984,E2 17362.984} C_VEL
LIN {X 0,Y 360.788,Z 1123.936,A -85,B 0,C 180,E1 17359.299,E2 17359.299} C_VEL
LIN {X 0,Y 361.854,Z 1119.208,A -85,B 0,C 180,E1 17355.907,E2 17355.907} C_VEL
LIN {X 0,Y 363.905,Z 1112.109,A -85,B 0,C 180,E1 17352.077,E2 17352.077} C_VEL
LIN {X 0,Y 366.575,Z 1104.309,A -85,B 0,C 180,E1 17348.729,E2 17348.729} C_VEL
LIN {X 0,Y 370.336,Z 1094.304,A -85,B 0,C 180,E1 17345.26,E2 17345.26} C_VEL
LIN {X 0,Y 375.007,Z 1082.826,A -85,B 0,C 180,E1 17341.953,E2 17341.953} C_VEL
LIN {X 0,Y 380.195,Z 1070.226,A -85,B 0,C 180,E1 17338.971,E2 17338.971} C_VEL
LIN {X 0,Y 385.712,Z 1057.095,A -85,B 0,C 180,E1 17336.313,E2 17336.313} C_VEL
LIN {X 0,Y 386.829,Z 1052.616,A -85,B 0,C 180,E1 17335.386,E2 17335.386} C_VEL
LIN {X 0,Y 386.711,Z 1041.18,A -85,B 0,C 180,E1 17332.931,E2 17332.931} C_VEL
LIN {X 0,Y 387.935,Z 1036.089,A -85,B 0,C 180,E1 17332.084,E2 17332.084} C_VEL
LIN {X 0,Y 394.546,Z 1019.485,A -85,B 0,C 180,E1 17329.836,E2 17329.836} C_VEL
LIN {X 0,Y 401.461,Z 1001.239,A -85,B 0,C 180,E1 17327.742,E2 17327.742} C_VEL
LIN {X 0,Y 407.858,Z 982.723,A -85,B 0,C 180,E1 17325.971,E2 17325.971} C_VEL
LIN {X 0,Y 414.405,Z 962.053,A -85,B 0,C 180,E1 17324.319,E2 17324.319} C_VEL
LIN {X 0,Y 419.625,Z 943.407,A -85,B 0,C 180,E1 17323.085,E2 17323.085} C_VEL
LIN {X 0,Y 425.05,Z 921.411,A -85,B 0,C 180,E1 17321.88,E2 17321.88} C_VEL
LIN {X 0,Y 429.221,Z 901.142,A -85,B 0,C 180,E1 17320.994,E2 17320.994} C_VEL
LIN {X 0,Y 433.157,Z 877.991,A -85,B 0,C 180,E1 17320.195,E2 17320.195} C_VEL
LIN {X 0,Y 435.96,Z 855.704,A -85,B 0,C 180,E1 17319.634,E2 17319.634} C_VEL
LIN {X 0,Y 438.12,Z 827.65,A -85,B 0,C 180,E1 17319.124,E2 17319.124} C_VEL
LIN {X 0,Y 451.643,Z 594.29,A -85,B 0,C 180,E1 17315.412,E2 17315.412} C_VEL
LIN {X 0,Y 443.11,Z 578.631,A -85,B 0,C 180,E1 17313.253,E2 17313.253} C_VEL
LIN {X 0,Y 434.431,Z 563.644,A -85,B 0,C 180,E1 17310.843,E2 17310.843} C_VEL
LIN {X 0,Y 426.523,Z 551.127,A -85,B 0,C 180,E1 17308.417,E2 17308.417} C_VEL
LIN {X 0,Y 420.674,Z 542.181,A -85,B 0,C 180,E1 17306.428,E2 17306.428} C_VEL
LIN {X 0,Y 413.126,Z 531.117,A -85,B 0,C 180,E1 17303.538,E2 17303.538} C_VEL
LIN {X 0,Y 408.621,Z 524.881,A -85,B 0,C 180,E1 17301.579,E2 17301.579} C_VEL
LIN {X 0,Y 402.842,Z 516.789,A -85,B 0,C 180,E1 17298.675,E2 17298.675} C_VEL
LIN {X 0,Y 399.195,Z 511.916,A -85,B 0,C 180,E1 17296.517,E2 17296.517} C_VEL
LIN {X 0,Y 394.603,Z 505.972,A -85,B 0,C 180,E1 17293.183,E2 17293.183} C_VEL
LIN {X 0,Y 390.818,Z 500.716,A -85,B 0,C 180,E1 17289.276,E2 17289.276} C_VEL
LIN {X 0,Y 388.08,Z 497.183,A -85,B 0,C 180,E1 17283.249,E2 17283.249} C_VEL
LIN {X 0,Y 388.26,Z 496.796,A -85,B 0,C 180,E1 17279.705,E2 17279.705} C_VEL
LIN {X 0,Y 389.714,Z 498.25,A -85,B 0,C 180,E1 17276.175,E2 17276.175} C_VEL
LIN {X 0,Y 394.426,Z 502.849,A -85,B 0,C 180,E1 17270.884,E2 17270.884} C_VEL
LIN {X 0,Y 399.819,Z 509.047,A -85,B 0,C 180,E1 17266.993,E2 17266.993} C_VEL
LIN {X 0,Y 404.97,Z 515.212,A -85,B 0,C 180,E1 17264.094,E2 17264.094} C_VEL
LIN {X 0,Y 410.202,Z 521.776,A -85,B 0,C 180,E1 17261.599,E2 17261.599} C_VEL
LIN {X 0,Y 416.43,Z 529.685,A -85,B 0,C 180,E1 17259.037,E2 17259.037} C_VEL
LIN {X 0,Y 423.669,Z 539.49,A -85,B 0,C 180,E1 17256.42,E2 17256.42} C_VEL
LIN {X 0,Y 433.013,Z 552.833,A -85,B 0,C 180,E1 17253.46,E2 17253.46} C_VEL
LIN {X 0,Y 442.192,Z 567.084,A -85,B 0,C 180,E1 17250.874,E2 17250.874} C_VEL
LIN {X 0,Y 451.637,Z 582.938,A -85,B 0,C 180,E1 17248.463,E2 17248.463} C_VEL
LIN {X 0,Y 453.386,Z 586.364,A -85,B 0,C 180,E1 17248.03,E2 17248.03} C_VEL
LIN {X 0,Y 439.191,Z 812.41,A -85,B 0,C 180,E1 17244.273,E2 17244.273} C_VEL
LIN {X 0,Y 436.584,Z 849.278,A -85,B 0,C 180,E1 17243.613,E2 17243.613} C_VEL
LIN {X 0,Y 433.752,Z 872.315,A -85,B 0,C 180,E1 17243.039,E2 17243.039} C_VEL
LIN {X 0,Y 430.076,Z 895.414,A -85,B 0,C 180,E1 17242.29,E2 17242.29} C_VEL
LIN {X 0,Y 425.652,Z 917.419,A -85,B 0,C 180,E1 17241.359,E2 17241.359} C_VEL
LIN {X 0,Y 420.61,Z 939.293,A -85,B 0,C 180,E1 17240.227,E2 17240.227} C_VEL
LIN {X 0,Y 414.743,Z 961.023,A -85,B 0,C 180,E1 17238.84,E2 17238.84} C_VEL
LIN {X 0,Y 408.765,Z 981.137,A -85,B 0,C 180,E1 17237.313,E2 17237.313} C_VEL
LIN {X 0,Y 402.153,Z 1001.239,A -85,B 0,C 180,E1 17235.48,E2 17235.48} C_VEL
LIN {X 0,Y 395.914,Z 1018.957,A -85,B 0,C 180,E1 17233.588,E2 17233.588} C_VEL
LIN {X 0,Y 388.77,Z 1038.031,A -85,B 0,C 180,E1 17231.179,E2 17231.179} C_VEL
LIN {X 0,Y 382.648,Z 1053.786,A -85,B 0,C 180,E1 17228.84,E2 17228.84} C_VEL
LIN {X 0,Y 375.823,Z 1070.974,A -85,B 0,C 180,E1 17225.826,E2 17225.826} C_VEL
LIN {X 0,Y 370.473,Z 1084.464,A -85,B 0,C 180,E1 17223.038,E2 17223.038} C_VEL
LIN {X 0,Y 364.946,Z 1098.716,A -85,B 0,C 180,E1 17219.549,E2 17219.549} C_VEL
LIN {X 0,Y 360.878,Z 1109.842,A -85,B 0,C 180,E1 17216.316,E2 17216.316} C_VEL
LIN {X 0,Y 357.274,Z 1120.652,A -85,B 0,C 180,E1 17212.546,E2 17212.546} C_VEL
LIN {X 0,Y 355.013,Z 1128.493,A -85,B 0,C 180,E1 17209.24,E2 17209.24} C_VEL
LIN {X 0,Y 353.237,Z 1136.154,A -85,B 0,C 180,E1 17205.263,E2 17205.263} C_VEL
LIN {X 0,Y 352.386,Z 1141.297,A -85,B 0,C 180,E1 17201.78,E2 17201.78} C_VEL
LIN {X 0,Y 352.023,Z 1145.145,A -85,B 0,C 180,E1 17198.329,E2 17198.329} C_VEL
LIN {X 0,Y 351.949,Z 1147.787,A -85,B 0,C 180,E1 17194.563,E2 17194.563} C_VEL
LIN {X 0,Y 351.968,Z 1148.797,A -85,B 0,C 180,E1 17191.465,E2 17191.465} C_VEL
LIN {X 0,Y 351.968,Z 1148.795,A -85,B 0,C 180,E1 17188.535,E2 17188.535} C_VEL
LIN {X 0,Y 351.94,Z 1147.637,A -85,B 0,C 180,E1 17185.111,E2 17185.111} C_VEL
LIN {X 0,Y 352.053,Z 1144.796,A -85,B 0,C 180,E1 17181.342,E2 17181.342} C_VEL
LIN {X 0,Y 352.413,Z 1141.05,A -85,B 0,C 180,E1 17178.046,E2 17178.046} C_VEL
LIN {X 0,Y 353.41,Z 1135.325,A -85,B 0,C 180,E1 17174.24,E2 17174.24} C_VEL
LIN {X 0,Y 355.105,Z 1128.087,A -85,B 0,C 180,E1 17170.594,E2 17170.594} C_VEL
LIN {X 0,Y 357.544,Z 1119.772,A -85,B 0,C 180,E1 17167.125,E2 17167.125} C_VEL
LIN {X 0,Y 361.24,Z 1108.728,A -85,B 0,C 180,E1 17163.358,E2 17163.358} C_VEL
LIN {X 0,Y 365.396,Z 1097.474,A -85,B 0,C 180,E1 17160.13,E2 17160.13} C_VEL
LIN {X 0,Y 370.739,Z 1083.659,A -85,B 0,C 180,E1 17156.804,E2 17156.804} C_VEL
LIN {X 0,Y 376.127,Z 1070.085,A -85,B 0,C 180,E1 17154.02,E2 17154.02} C_VEL
LIN {X 0,Y 382.699,Z 1053.493,A -85,B 0,C 180,E1 17151.132,E2 17151.132} C_VEL
LIN {X 0,Y 388.753,Z 1037.888,A -85,B 0,C 180,E1 17148.818,E2 17148.818} C_VEL
LIN {X 0,Y 396.111,Z 1018.16,A -85,B 0,C 180,E1 17146.339,E2 17146.339} C_VEL
LIN {X 0,Y 402.237,Z 1000.721,A -85,B 0,C 180,E1 17144.485,E2 17144.485} C_VEL
LIN {X 0,Y 409.468,Z 978.421,A -85,B 0,C 180,E1 17142.484,E2 17142.484} C_VEL
LIN {X 0,Y 415.094,Z 959.438,A -85,B 0,C 180,E1 17141.065,E2 17141.065} C_VEL
LIN {X 0,Y 421.197,Z 936.299,A -85,B 0,C 180,E1 17139.622,E2 17139.622} C_VEL
LIN {X 0,Y 425.905,Z 915.721,A -85,B 0,C 180,E1 17138.576,E2 17138.576} C_VEL
LIN {X 0,Y 430.588,Z 891.671,A -85,B 0,C 180,E1 17137.592,E2 17137.592} C_VEL
LIN {X 0,Y 433.892,Z 870.468,A -85,B 0,C 180,E1 17136.923,E2 17136.923} C_VEL
LIN {X 0,Y 436.769,Z 846.078,A -85,B 0,C 180,E1 17136.333,E2 17136.333} C_VEL
LIN {X 0,Y 440.924,Z 782.138,A -85,B 0,C 180,E1 17135.234,E2 17135.234} C_VEL
LIN {X 0,Y 453.24,Z 585.994,A -85,B 0,C 180,E1 17131.969,E2 17131.969} C_VEL
LIN {X 0,Y 444.797,Z 571.469,A -85,B 0,C 180,E1 17129.863,E2 17129.863} C_VEL
LIN {X 0,Y 435.317,Z 556.39,A -85,B 0,C 180,E1 17127.274,E2 17127.274} C_VEL
LIN {X 0,Y 425.832,Z 542.591,A -85,B 0,C 180,E1 17124.373,E2 17124.373} C_VEL
LIN {X 0,Y 418.183,Z 532.128,A -85,B 0,C 180,E1 17121.717,E2 17121.717} C_VEL
LIN {X 0,Y 411.522,Z 523.429,A -85,B 0,C 180,E1 17119.075,E2 17119.075} C_VEL
LIN {X 0,Y 407.056,Z 517.945,A -85,B 0,C 180,E1 17117.07,E2 17117.07} C_VEL
LIN {X 0,Y 403.298,Z 513.253,A -85,B 0,C 180,E1 17115.163,E2 17115.163} C_VEL
LIN {X 0,Y 398.683,Z 507.753,A -85,B 0,C 180,E1 17112.456,E2 17112.456} C_VEL
LIN {X 0,Y 393.578,Z 501.946,A -85,B 0,C 180,E1 17108.621,E2 17108.621} C_VEL
LIN {X 0,Y 388.862,Z 497.262,A -85,B 0,C 180,E1 17102.8,E2 17102.8} C_VEL
LIN {X 0,Y 387.769,Z 496.274,A -85,B 0,C 180,E1 17099.261,E2 17099.261} C_VEL
LIN {X 0,Y 387.893,Z 497.105,A -85,B 0,C 180,E1 17095.861,E2 17095.861} C_VEL
LIN {X 0,Y 391.104,Z 501.137,A -85,B 0,C 180,E1 17089.914,E2 17089.914} C_VEL
LIN {X 0,Y 395.471,Z 507.198,A -85,B 0,C 180,E1 17085.803,E2 17085.803} C_VEL
LIN {X 0,Y 399.249,Z 512.134,A -85,B 0,C 180,E1 17083.186,E2 17083.186} C_VEL
LIN {X 0,Y 404.515,Z 519.253,A -85,B 0,C 180,E1 17080.206,E2 17080.206} C_VEL
LIN {X 0,Y 410.536,Z 527.59,A -85,B 0,C 180,E1 17077.367,E2 17077.367} C_VEL
LIN {X 0,Y 416.767,Z 536.574,A -85,B 0,C 180,E1 17074.833,E2 17074.833} C_VEL
LIN {X 0,Y 423.384,Z 546.278,A -85,B 0,C 180,E1 17072.465,E2 17072.465} C_VEL
LIN {X 0,Y 431.773,Z 559.382,A -85,B 0,C 180,E1 17069.794,E2 17069.794} C_VEL
LIN {X 0,Y 441.554,Z 575.929,A -85,B 0,C 180,E1 17067.021,E2 17067.021} C_VEL
LIN {X 0,Y 450.956,Z 593.167,A -85,B 0,C 180,E1 17064.621,E2 17064.621} C_VEL
LIN {X 0,Y 451.482,Z 594.562,A -85,B 0,C 180,E1 17064.482,E2 17064.482} C_VEL
LIN {X 0,Y 437.191,Z 840.191,A -85,B 0,C 180,E1 17060.563,E2 17060.563} C_VEL
LIN {X 0,Y 435.053,Z 862.868,A -85,B 0,C 180,E1 17060.104,E2 17060.104} C_VEL
LIN {X 0,Y 431.7,Z 886.299,A -85,B 0,C 180,E1 17059.438,E2 17059.438} C_VEL
LIN {X 0,Y 427.761,Z 908.213,A -85,B 0,C 180,E1 17058.62,E2 17058.62} C_VEL
LIN {X 0,Y 422.789,Z 930.42,A -85,B 0,C 180,E1 17057.551,E2 17057.551} C_VEL
LIN {X 0,Y 417.207,Z 952.077,A -85,B 0,C 180,E1 17056.269,E2 17056.269} C_VEL
LIN {X 0,Y 411.281,Z 971.808,A -85,B 0,C 180,E1 17054.833,E2 17054.833} C_VEL
LIN {X 0,Y 404.772,Z 991.648,A -85,B 0,C 180,E1 17053.11,E2 17053.11} C_VEL
LIN {X 0,Y 398.32,Z 1009.417,A -85,B 0,C 180,E1 17051.252,E2 17051.252} C_VEL
LIN {X 0,Y 391.445,Z 1027.23,A -85,B 0,C 180,E1 17049.056,E2 17049.056} C_VEL
LIN {X 0,Y 385.225,Z 1042.316,A -85,B 0,C 180,E1 17046.84,E2 17046.84} C_VEL
LIN {X 0,Y 378.785,Z 1057.589,A -85,B 0,C 180,E1 17044.213,E2 17044.213} C_VEL
LIN {X 0,Y 373.067,Z 1070.716,A -85,B 0,C 180,E1 17041.509,E2 17041.509} C_VEL
LIN {X 0,Y 367.599,Z 1083.459,A -85,B 0,C 180,E1 17038.425,E2 17038.425} C_VEL
LIN {X 0,Y 363.033,Z 1094.213,A -85,B 0,C 180,E1 17035.272,E2 17035.272} C_VEL
